    // --- All valves confirmed off
    logs.M_LogInfo('LN2 filling stopped successfully.');
    M_Activity_Stop_LN2_Filling := TRUE;
    TurningOFFTimeout(IN := FALSE);
    bAttemptingTurnOFF := FALSE;
    RETURN;
ELSE
    // --- Timeout expired: check what remains active
    IF lc_ln2_level_ctrl[1].LN2_Valve.stat.bActive THEN
        logs.M_LogInfo('LN2 shutdown timeout – Valve 1 still active');
        M_SetError(E1207_LN2_SHUTDOWN_V1_FAILED, 'LN2 Valve 1 failed to turn off');
    END_IF
    IF lc_ln2_level_ctrl[2].LN2_Valve.stat.bActive THEN
        logs.M_LogInfo('LN2 shutdown timeout – Valve 2 still active');
        M_SetError(E1208_LN2_SHUTDOWN_V2_FAILED, 'LN2 Valve 2 failed to turn off');
    END_IF
    IF lc_ln2_level_ctrl[3].LN2_Valve.stat.bActive THEN
        logs.M_LogInfo('LN2 shutdown timeout – Valve 3 still active');
        M_SetError(E1209_LN2_SHUTDOWN_V3_FAILED, 'LN2 Valve 3 failed to turn off');
    END_IF

    IF lc_ln2_level_ctrl[1].LN2_Valve.stat.bActive
    OR lc_ln2_level_ctrl[2].LN2_Valve.stat.bActive
    OR lc_ln2_level_ctrl[3].LN2_Valve.stat.bActive THEN
        M_SetError(E1206_LN2_Level_ShutdownTimeout, 'LN2 shutdown timeout: one or more valves still active');
        TurningOFFTimeout(IN := FALSE);
        bAttemptingTurnOFF := FALSE;
        M_Activity_Stop_LN2_Filling := FALSE;
        RETURN;
    ELSE
        logs.M_LogInfo('LN2 filling turned off successfully (after timeout).');
        M_Activity_Stop_LN2_Filling := TRUE;
        TurningOFFTimeout(IN := FALSE);
        bAttemptingTurnOFF := FALSE;
        RETURN;
    END_IF
END_IF
END_METHOD

METHOD M_Activity_Stop_PTCs : BOOL
VAR_INPUT
END_VAR
VAR_INST
    bErrorCond            : BOOL := FALSE;
    bAttemptingTurnOFF    : BOOL := FALSE;

    TurningOFFTimeout     : TON;
    tTurningOFFTime       : TIME := T#10M;
END_VAR
//  Start shutdown process 
IF NOT bAttemptingTurnOFF THEN
    bAttemptingTurnOFF := TRUE;
    logs.M_LogInfo('Initiating PTC shutdown...');
    
    TurningOFFTimeout(IN := TRUE, PT := tTurningOFFTime);
	ctrl.bPTC_1_Enable := FALSE;
	ctrl.bPTC_2_Enable := FALSE;
	ctrl.bPTC_3_Enable := FALSE;
END_IF

// Wait for confirmation of shutdown or timeout
IF NOT TurningOFFTimeout.Q THEN
    IF ptc[1].stat.bSystemOn OR ptc[2].stat.bSystemOn OR ptc[3].stat.bSystemOn THEN
        M_Activity_Stop_PTCs := FALSE;
        RETURN;
    END_IF

    // All PTCs confirmed off
    logs.M_LogInfo('PTCs successfully turned off.');
    M_Activity_Stop_PTCs := TRUE;
    TurningOFFTimeout(IN := FALSE);
    bAttemptingTurnOFF := FALSE;
    RETURN;
ELSE
    // Timeout expired — check if PTC or PTCs are still active
    IF ptc[1].stat.bSystemOn OR ptc[2].stat.bSystemOn OR ptc[3].stat.bSystemOn THEN
        logs.M_LogInfo('PTC shutdown timeout – one or more PTCs failed to stop.');
        M_SetError(E1907_PTC_ShutdownTimeout, 'PTC shutdown timeout: at least one PTC still active.');
        TurningOFFTimeout(IN := FALSE);
        bAttemptingTurnOFF := FALSE;
        M_Activity_Stop_PTCs := FALSE;
        RETURN;
    ELSE
        logs.M_LogInfo('PTCs turned off successfully (after timeout).');
        M_Activity_Stop_PTCs := TRUE;
        TurningOFFTimeout(IN := FALSE);
        bAttemptingTurnOFF := FALSE;
        RETURN;
    END_IF
END_IF
END_METHOD

METHOD M_Activity_Stopping_Cool_Down : BOOL
VAR_INPUT
END_VAR
VAR_IN_OUT
	{attribute 'OPC.UA.DA' := '0'}
	all_cryo_temps:					FB_METIS_TEMPERATURES;
	{attribute 'OPC.UA.DA' := '0'}
	all_heaters:					FB_METIS_HEATERS;
	{attribute 'OPC.UA.DA' := '0'}
	all_t_ctrls:      				FB_METIS_TCTRL;
	{attribute 'OPC.UA.DA' := '0'}
	all_t_votes: 					FB_METIS_VOTERS;
	{attribute 'OPC.UA.DA' := '0'}
	interlocks:						T_METIS_CRYO_INTERLOCKS;
END_VAR
VAR_INST
    StopCooldownAttempts : UINT := 0;
    MaxStopCooldownAttempts : UINT := 3; 
END_VAR
CASE stat.nStopCoolDownState OF

// Check readiness 
0:
    logs.M_LogInfo('Stopping cooldown: checking if system is ready for operation...');
    
    IF stat.bReadyForOperations THEN
		
		stat.bPermitEvacuationStop := TRUE;
        M_PermitEvacuationStop();
        logs.M_LogInfo('System is cold and ready – evacuation stop permitted.');
        stat.nStopCoolDownState := 50;

    ELSE
		stat.bPermitEvacuationStop := FALSE;
        logs.M_LogInfo('System is not cold – evacuation stop blocked.');
		// stat.nState := E_MET_CRYO_COOLDOWN_STATE.KEEP_COOLING;
		//M_Activity_Stopping_Cool_Down := FALSE;
        stat.nStopCoolDownState := 50;
    END_IF
    

// Declare Cooldown Finished
50:
    logs.M_LogInfo('Cooldown process finished.');
    stat.nState := E_MET_CRYO_COOLDOWN_STATE.FINISHED;
    stat.nStopCoolDownState := 0; 
    M_Activity_Stopping_Cool_Down := TRUE;
    RETURN;

// Error state 
99:
    logs.M_LogInfo('Cooldown stop failed. Entered error fallback.');
    stat.nState := E_MET_CRYO_COOLDOWN_STATE.ERROR;
    M_Activity_Stopping_Cool_Down := FALSE;
    RETURN;

END_CASE

M_Activity_Stopping_Cool_Down := FALSE;
END_METHOD

METHOD M_Check_Is_ReadyForOperation : BOOL
VAR_INPUT
END_VAR
VAR_IN_OUT
	{attribute 'OPC.UA.DA' := '0'}
	all_cryo_temps:					FB_METIS_TEMPERATURES;
	{attribute 'OPC.UA.DA' := '0'}
	all_heaters:					FB_METIS_HEATERS;
	{attribute 'OPC.UA.DA' := '0'}
	all_t_ctrls:      				FB_METIS_TCTRL;
	{attribute 'OPC.UA.DA' := '0'}
	all_t_votes: 					FB_METIS_VOTERS;
	{attribute 'OPC.UA.DA' := '0'}
	interlocks:						T_METIS_CRYO_INTERLOCKS;
END_VAR
// Check if the system is ready for operations (all temps achieved)




IF in_Cryo_Stat.bInGoodVacuum AND in_Cryo_Stat.lrRadiationShieldsTempK <  100.0 AND in_Cryo_Stat.lrHighestTempK < 75.0 THEN
	stat.bReadyForOperations := TRUE;
ELSE
	stat.bReadyForOperations := FALSE;
END_IF
END_METHOD

METHOD M_Check_LN2_Filling_Status : BOOL
VAR_INPUT
END_VAR
VAR_INST
	bLN2_FillingError :		BOOL := TRUE;
	bAttemptingRecovery:	BOOL := FALSE;
	RecoveryTimeout:		TON;
	tRecoveryTime:			TIME := T#30S;
END_VAR
// precondition checks

bLN2_FillingError := FALSE;

IF NOT in_Cryo_Stat.bEvacuationActive THEN
    IF NOT bLN2_FillingError THEN
        M_SetError(E1004_PumpsNotRunning, 'Evacuation is not active');
        bLN2_FillingError := TRUE;
    END_IF
ELSIF NOT bESO_LN2_Supply THEN
    IF NOT bLN2_FillingError THEN
        M_SetError(E1005_LN2SupplyNotReady, 'LN2 supply unavailable');
        bLN2_FillingError := TRUE;
    END_IF
END_IF

// Valve error checks
IF lc_ln2_level_ctrl[1].LN2_Valve.stat.bError THEN
    M_SetError(E1100_SHA_V_Error, 'Error in LN2 Valve – Stiff Ring');
    bLN2_FillingError := TRUE;
ELSIF lc_ln2_level_ctrl[2].LN2_Valve.stat.bError THEN
    M_SetError(E1101_SHB_V_Error, 'Error in LN2 Valve – Middle Segment');
    bLN2_FillingError := TRUE;
ELSIF lc_ln2_level_ctrl[3].LN2_Valve.stat.bError THEN
    M_SetError(E1102_SHC_V_Error, 'Error in LN2 Valve – Lower Segment');
    bLN2_FillingError := TRUE;
END_IF

//IF NOT lc_ln2_level_ctrl[1].bActive OR NOT lc_ln2_level_ctrl[2].bActive OR NOT lc_ln2_level_ctrl[3].bActive THEN
//	 bLN2_FillingError := TRUE;
//END_IF

// Recoverying
IF NOT bLN2_FillingError THEN
	
	// All is good
	RecoveryTimeout(IN := FALSE);
	bAttemptingRecovery := FALSE;
	bLN2_FillingError := FALSE;
	M_Check_LN2_Filling_Status := TRUE;
	RETURN;
ELSE

    IF NOT bAttemptingRecovery THEN
        bAttemptingRecovery := TRUE;
        RecoveryTimeout(IN := TRUE, PT := tRecoveryTime);
		logs.M_LogInfo('Error LN2 Filling: Recovering...');
		ctrl.bEnable_LN2_Level_Control[1] := FALSE;
		ctrl.bEnable_LN2_Level_Control[2] := FALSE;
		ctrl.bEnable_LN2_Level_Control[3] := FALSE;
		lc_ln2_level_ctrl[1].LN2_Valve.M_Reset();
        lc_ln2_level_ctrl[2].LN2_Valve.M_Reset();
        lc_ln2_level_ctrl[3].LN2_Valve.M_Reset();
		lc_ln2_level_ctrl[1].M_Reset();
		lc_ln2_level_ctrl[2].M_Reset();
		lc_ln2_level_ctrl[3].M_Reset();
    END_IF

    IF NOT RecoveryTimeout.Q THEN
		ctrl.bEnable_LN2_Level_Control[1] := TRUE;
		ctrl.bEnable_LN2_Level_Control[2] := TRUE;
		ctrl.bEnable_LN2_Level_Control[3] := TRUE;
		RecoveryTimeout(IN := TRUE, PT := tRecoveryTime);
    ELSE
        // Recovery failed → shutdown filling
        ctrl.bEnable_LN2_Level_Control[1] := FALSE;
        ctrl.bEnable_LN2_Level_Control[2] := FALSE;
        ctrl.bEnable_LN2_Level_Control[3] := FALSE;
        tDelay_SHB(IN := FALSE);
        tDelay_SHC(IN := FALSE);
        stat.nState := E_MET_CRYO_COOLDOWN_STATE.ERROR;
        stat.sState := 'LN2 Filling Failed – Recovery Timeout';
		logs.M_LogInfo('LN2 Filling Failed – Recovery Timeout');
        RecoveryTimeout(IN := FALSE);
        bAttemptingRecovery := FALSE;
    END_IF

    M_Check_LN2_Filling_Status := FALSE;
    RETURN;
END_IF
END_METHOD

METHOD M_Check_PTCs_Heater_Ctrl_Status : BOOL
VAR_INPUT
END_VAR
VAR_INST
    bErrorCond           : BOOL := FALSE;
    bAttemptingRecovery  : BOOL := FALSE;	
END_VAR
VAR_IN_OUT
	{attribute 'OPC.UA.DA' := '0'}
	all_cryo_temps:					FB_METIS_TEMPERATURES;
	{attribute 'OPC.UA.DA' := '0'}
	all_heaters:					FB_METIS_HEATERS;
	{attribute 'OPC.UA.DA' := '0'}
	all_t_ctrls:      				FB_METIS_TCTRL;
	{attribute 'OPC.UA.DA' := '0'}
	all_t_votes: 					FB_METIS_VOTERS;
	{attribute 'OPC.UA.DA' := '0'}
	interlocks:						T_METIS_CRYO_INTERLOCKS;
END_VAR


IF 	all_heaters.h_cry_pta.stat.bError THEN
	M_SetError(E1308_EarFlange_TempCtrlFault, 'h_cry_pta in error...');
    bErrorCond := TRUE;
END_IF

IF 	all_heaters.h_cry_ptb.stat.bError THEN
	M_SetError(E1308_EarFlange_TempCtrlFault, 'h_cry_ptb in error...');
    bErrorCond := TRUE;
END_IF

IF 	all_heaters.h_cry_ptc.stat.bError THEN
	M_SetError(E1308_EarFlange_TempCtrlFault, 'h_cry_ptc in error...');
    bErrorCond := TRUE;
END_IF

IF 	all_t_ctrls.tc_cry_pt.stat.bError THEN
	M_SetError(E1308_EarFlange_TempCtrlFault, 'tc_cry_pt temp ctrl in error...');
    bErrorCond := TRUE;
END_IF


IF bErrorCond THEN
	
	M_Check_PTCs_Heater_Ctrl_Status := FALSE;
	logs.M_LogInfo('Temp Ctrl anomaly at stiff ring');
	stat.bWarning := TRUE;
    RETURN;
	
END_IF


M_Check_PTCs_Heater_Ctrl_Status := TRUE;
END_METHOD

METHOD M_Check_PTCs_Status : BOOL
VAR_INPUT
END_VAR
VAR_INST
    bErrorCond           : BOOL := FALSE;
    bAttemptingRecovery  : BOOL := FALSE;

    RecoveryTimeout      : TON;
    tRecoveryTime        : TIME := T#10M;

    ToggleTimeoutPTC1    : TON;
    ToggleTimeoutPTC2    : TON;
    ToggleTimeoutPTC3    : TON;
    tToggleTime          : TIME := T#5M;

    bTogglePTC1          : BOOL := FALSE;
    bTogglePTC2          : BOOL := FALSE;
    bTogglePTC3          : BOOL := FALSE;
END_VAR


// Check PTC Active Status
bErrorCond := FALSE;

IF NOT ptc[1].stat.bActive THEN
    M_SetError(E1903_PTC1_NotActive, 'PTC 1 not active');
    bErrorCond := TRUE;
END_IF

IF NOT ptc[2].stat.bActive THEN
    M_SetError(E1904_PTC2_NotActive, 'PTC 2 not active');
    bErrorCond := TRUE;
END_IF

IF NOT ptc[3].stat.bActive THEN
    M_SetError(E1905_PTC3_NotActive, 'PTC 3 not active');
    bErrorCond := TRUE;
END_IF

IF NOT bErrorCond THEN
    RecoveryTimeout		(IN := FALSE);
    ToggleTimeoutPTC1	(IN := FALSE);
    ToggleTimeoutPTC2	(IN := FALSE);
    ToggleTimeoutPTC3	(IN := FALSE);
    bAttemptingRecovery := FALSE;
    M_Check_PTCs_Status := TRUE;
    RETURN;
END_IF

// Handle Recovery
IF NOT bAttemptingRecovery THEN
    bAttemptingRecovery := TRUE;
    RecoveryTimeout(IN := TRUE, PT := tRecoveryTime);
    logs.M_LogInfo('PTC failure detected: entering recovery...');
END_IF

IF NOT RecoveryTimeout.Q THEN

    //  PTC 1 Recovery Toggle
    IF NOT ptc[1].stat.bActive THEN
        ToggleTimeoutPTC1(IN := TRUE, PT := tToggleTime);
        IF ToggleTimeoutPTC1.Q THEN
            IF bTogglePTC1 THEN
                ptc[1].in_bEnable := TRUE;
            ELSE
                ptc[1].in_bEnable := FALSE;
            END_IF
            bTogglePTC1 := NOT bTogglePTC1;
            ToggleTimeoutPTC1(IN := FALSE); // Restart toggle delay
        END_IF
    ELSE
        ToggleTimeoutPTC1(IN := FALSE);
    END_IF

    // PTC 2 Recovery Toggle
    IF NOT ptc[2].stat.bActive THEN
        ToggleTimeoutPTC2(IN := TRUE, PT := tToggleTime);
        IF ToggleTimeoutPTC2.Q THEN
            IF bTogglePTC2 THEN
                ptc[2].in_bEnable := TRUE;
            ELSE
                ptc[2].in_bEnable := FALSE;
            END_IF
            bTogglePTC2 := NOT bTogglePTC2;
            ToggleTimeoutPTC2(IN := FALSE);
        END_IF
    ELSE
        ToggleTimeoutPTC2(IN := FALSE);
    END_IF

    // PTC 3 Recovery Toggle
    IF NOT ptc[3].stat.bActive THEN
        ToggleTimeoutPTC3(IN := TRUE, PT := tToggleTime);
        IF ToggleTimeoutPTC3.Q THEN
            IF bTogglePTC3 THEN
                ptc[3].in_bEnable := TRUE;
            ELSE
                ptc[3].in_bEnable := FALSE;
            END_IF
            bTogglePTC3 := NOT bTogglePTC3;
            ToggleTimeoutPTC3(IN := FALSE);
        END_IF
    ELSE
        ToggleTimeoutPTC3(IN := FALSE);
    END_IF

    M_Check_PTCs_Status := FALSE;
    RETURN;
ELSE
    // Recovery Failed 
    ptc[1].in_bEnable := FALSE;
    ptc[2].in_bEnable := FALSE;
    ptc[3].in_bEnable := FALSE;

    stat.bWarning := TRUE;
    M_SetError(E1906_PTC_Failure, 'PTC recovery failed after timeout');
    stat.nState := E_MET_CRYO_COOLDOWN_STATE.STOPPING_COOL_DOWN;
    RecoveryTimeout(IN := FALSE);
    ToggleTimeoutPTC1(IN := FALSE);
    ToggleTimeoutPTC2(IN := FALSE);
    ToggleTimeoutPTC3(IN := FALSE);

    bAttemptingRecovery := FALSE;
    M_Check_PTCs_Status := FALSE;
END_IF
END_METHOD

METHOD M_Configure
VAR_INPUT
END_VAR

	////////////////////////
	// Pre-Cooling valves//
	//////////////////////



// Set pointers to Valves - MUST!!!
ptrV[1]	:= ADR(PVV_P1);
ptrV[2]	:= ADR(PVV_P2);
ptrV[3]	:= ADR(PVV_P3);


// Set pointers to Valve Commands - MUST!!!
ptrVC[1]	:= ADR(ctrl.cor_PVV_P1);
ptrVC[2]	:= ADR(ctrl.cor_PVV_P2);
ptrVC[3]	:= ADR(ctrl.cor_PVV_P3);


// Set pointers to Enable Valves flags - MUST!!!
ptrEV[1]	:= ADR(ctrl.bEnable_PVV_P1);
ptrEV[2]	:= ADR(ctrl.bEnable_PVV_P2);
ptrEV[3]	:= ADR(ctrl.bEnable_PVV_P3);



IF NOT bConfigured THEN


	bPwr_VAG_PCA 	:= TRUE;
	bPwr_VAG_PCB 	:= TRUE;      
	bPwr_VAG_P1 	:= TRUE;
	
	PVV_P1.M_Reset();
	PVV_P2.M_Reset();
	PVV_P3.M_Reset();
	
	///////////////////////
	///// PTC Coolers /////
	//////////////////////		

	// Set pointers to command override instances
	ptrArr_cor_ptcs[1] := ADR(ctrl.cor_PTC_1);
	ptrArr_cor_ptcs[2] := ADR(ctrl.cor_PTC_2);
	ptrArr_cor_ptcs[3] := ADR(ctrl.cor_PTC_3);
	
	
	////////////////////////////////
	// LN2 Level Sensors & Control//
	////////////////////////////////

	ctrl.bEnable_LN2_Level_Control[1] := FALSE;
	ctrl.bEnable_LN2_Level_Control[2] := FALSE;
	ctrl.bEnable_LN2_Level_Control[3] := FALSE; 
	
	
	// This call just configures logs at the very start.
	// Logging is done by explicit calls to M_LogInfo().
	logs(in_sName := in_sName);
	
	M_ResetValves();
	
	bConfigured := TRUE;

END_IF
END_METHOD

METHOD M_ExecuteControllers
VAR_INPUT
END_VAR
////////////////////////
// Pre-Cooling valves//
//////////////////////

//ctrl.bEnable_PVV_P1 := in_bEnable_PVV_P1;
ctrl.bEnable_PVV_P1 := TRUE; // TODO: Implement for EVAC and Pre-cooling
ctrl.bEnable_PVV_P2 := in_bEnable_PVV_P2;
ctrl.bEnable_PVV_P3 := in_bEnable_PVV_P3;

// Valve commands
ctrl.cor_PVV_P1(in_bEnable := ctrl.bEnable_PVV_P1);	// Handling of PVV_P1 commands
ctrl.cor_PVV_P2(in_bEnable := ctrl.bEnable_PVV_P2);	// Handling of PVV_P2 commands
ctrl.cor_PVV_P3(in_bEnable := ctrl.bEnable_PVV_P3);	// Handling of PVV_P3 commands

// Valve Control
IF PVV_P1.stat.bError THEN
	PVV_P1.M_Reset();
END_IF 
PVV_P1(
	in_bEnable			:= ctrl.cor_PVV_P1.out_bEnable,
	in_nFeedback		:= E_CRYO_BIN_ACT_FEEDBACK.ON_AND_OFF);
	
PVV_P2(
	in_bEnable			:= ctrl.cor_PVV_P2.out_bEnable,
	in_nFeedback		:= E_CRYO_BIN_ACT_FEEDBACK.ON_AND_OFF);
	
PVV_P3(
	in_bEnable			:= ctrl.cor_PVV_P3.out_bEnable,
	in_nFeedback		:= E_CRYO_BIN_ACT_FEEDBACK.ON_AND_OFF);


///////////////////////
// LN2 Level Sensors//
//////////////////////



lc_ln2_level_ctrl[1](in_sName := 'Stiff_Ring',
					in_bEnable:= ctrl.bEnable_LN2_Level_Control[1], 
					in_ESO_LN2_Supply := bESO_LN2_Supply,
					in_bEarly_Refilling:= FALSE);
	
lc_ln2_level_ctrl[2](in_sName := 'Intermediate_Segment',
					in_bEnable:= ctrl.bEnable_LN2_Level_Control[2], 
					in_ESO_LN2_Supply := bESO_LN2_Supply,
					in_bEarly_Refilling:= FALSE);

lc_ln2_level_ctrl[3](in_sName := 'Bottom_Segment',
					in_bEnable:= ctrl.bEnable_LN2_Level_Control[3], 
					in_ESO_LN2_Supply := bESO_LN2_Supply,
					in_bEarly_Refilling:= FALSE);
	
	
///////////////////////
///// PTC Coolers /////
//////////////////////	

{IF defined (V1_HW)}
	
ctrl.cor_PTC_1(in_bEnable:=ctrl.bPTC_1_Enable);
ptc[1](
	in_bEnable:= ctrl.cor_PTC_1.out_bEnable,
	in_bSimulation:= FALSE, 
	in_sName:= 'PTC_A', 
	in_sSN_Compressor:= 'CPA286IW-19880300001', 
	in_sSN_PulseTube:= 'PT810-19880200001', 
	in_nYear_Compressor:= 2023, 
	in_nYear_PulseTube:= 2023, 
	in_lrNextService_Compressor:= 20000.0, 
	in_lrNextService_PulseTube:= 40000.0, 
	in_nSlaveID:= 16, 
	in_nPeriod:= 1000);
	

ctrl.cor_PTC_2(in_bEnable:=ctrl.bPTC_2_Enable);
ptc[2](
	in_bEnable:= ctrl.cor_PTC_2.out_bEnable,
	in_bSimulation:= FALSE, 
	in_sName:= 'PTC_B', 
	in_sSN_Compressor:= 'CPA286IW-19870300001', 
	in_sSN_PulseTube:= 'PT810-19870200001', 
	in_nYear_Compressor:= 2023, 
	in_nYear_PulseTube:= 2023, 
	in_lrNextService_Compressor:= 20000.0, 
	in_lrNextService_PulseTube:= 40000.0, 
	in_nSlaveID:= 16, 
	in_nPeriod:= 1000);
	

ctrl.cor_PTC_3(in_bEnable:=ctrl.bPTC_3_Enable);
ptc[3](
	in_bEnable:= ctrl.cor_PTC_3.out_bEnable,
	in_bSimulation:= FALSE, 
	in_sName:= 'PTC_C', 
	in_sSN_Compressor:= 'CPA286IW-19890300001', 
	in_sSN_PulseTube:= 'PT810-19890200001', 
	in_nYear_Compressor:= 2023, 
	in_nYear_PulseTube:= 2023, 
	in_lrNextService_Compressor:= 20000.0, 
	in_lrNextService_PulseTube:= 40000.0, 
	in_nSlaveID:= 16, 
	in_nPeriod:= 1000);

{END_IF}
 
{IF defined (V2_SIM)}	
	
ctrl.cor_PTC_1(in_bEnable:=ctrl.bPTC_1_Enable);
ptc[1](
	in_bEnable:= ctrl.cor_PTC_1.out_bEnable,
	in_bSimulation:= FALSE, 
	in_sName:= 'PTC_A', 
	in_sSN_Compressor:= 'CPA286IW-19880300001', 
	in_sSN_PulseTube:= 'PT810-19880200001', 
	in_nYear_Compressor:= 2023, 
	in_nYear_PulseTube:= 2023, 
	in_lrNextService_Compressor:= 20000.0, 
	in_lrNextService_PulseTube:= 40000.0, 
	in_nSlaveID:= 16, 
	in_nPeriod:= 1000);
	

ctrl.cor_PTC_2(in_bEnable:=ctrl.bPTC_2_Enable);
ptc[2](
	in_bEnable:= ctrl.cor_PTC_2.out_bEnable,
	in_bSimulation:= TRUE, 
	in_sName:= 'PTC_B', 
	in_sSN_Compressor:= 'CPA286IW-19870300001', 
	in_sSN_PulseTube:= 'PT810-19870200001', 
	in_nYear_Compressor:= 2023, 
	in_nYear_PulseTube:= 2023, 
	in_lrNextService_Compressor:= 20000.0, 
	in_lrNextService_PulseTube:= 40000.0, 
	in_nSlaveID:= 16, 
	in_nPeriod:= 1000);
	

ctrl.cor_PTC_3(in_bEnable:=ctrl.bPTC_3_Enable);
ptc[3](
	in_bEnable:= ctrl.cor_PTC_3.out_bEnable,
	in_bSimulation:= FALSE, 
	in_sName:= 'PTC_C', 
	in_sSN_Compressor:= 'CPA286IW-19890300001', 
	in_sSN_PulseTube:= 'PT810-19890200001', 
	in_nYear_Compressor:= 2023, 
	in_nYear_PulseTube:= 2023, 
	in_lrNextService_Compressor:= 20000.0, 
	in_lrNextService_PulseTube:= 40000.0, 
	in_nSlaveID:= 16, 
	in_nPeriod:= 1000);	
		
	
{END_IF}	
	
///////////////////////
///// ---------- /////
//////////////////////
END_METHOD

METHOD M_Get_ReadyForOperations : BOOL
VAR_INPUT
END_VAR
M_Get_ReadyForOperations := stat.bReadyForOperations;
END_METHOD

METHOD M_HandleEvents
VAR_INPUT
END_VAR

//
// Handle triggers
//

trigEnable	(CLK := ctrl.bEnable);
trigDisable	(CLK := ctrl.bEnable);
END_METHOD

METHOD M_HandleInterlocks
VAR_INPUT
END_VAR
//VAR_IN_OUT
//	{attribute 'OPC.UA.DA' := '0'}
//	interlocks:						T_METIS_CRYO_INTERLOCKS;
//END_VAR

//interlocks.bInterlock_Evacuation 			:= FALSE;
//interlocks.bInterlock_Venting 			:= TRUE; // Venting blocked
//interlocks.bInterlock_CoolDown 			:= FALSE; // Cool_Down, pre-cooling, LN2_filling blocked
//interlocks.bInterlock_WarmUp 				:= TRUE; // Warm_up Blocked
//interlocks.bInterlock_Regeneration 		:= TRUE;
//interlocks.bInterlock_AntiFogging 		:= FALSE;
//interlocks.bInterlock_PowerOutage 		:= FALSE;
//interlocks.bInterlock_StopPowerOutage		:= FALSE;

//interlocks.sInterlockState := 'COOL_DOWN Active';



//// Venting Valves Closed ---
//IF in_Cryo_Stat.bVentingValvesAreClosed THEN
//    stat.nState := E_MET_CRYO_VENTING_STATE.ERROR;
//    stat.sState := 'Error: Venting valves are closed.';
//    RETURN; 
//END_IF

//// Pumps Running ---
//IF in_Cryo_Stat.bPumpsAreRunning THEN
//    stat.nState := E_MET_CRYO_VENTING_STATE.ERROR;
//    stat.sState := 'Error: Pumps are Running.';
//    RETURN; 
//END_IF

//// --- Evacuation Activated ---
//IF in_Cryo_Stat.bEvacuationActive THEN
//    stat.nState := E_MET_CRYO_VENTING_STATE.ERROR;
//    stat.sState := 'Error: Evacuation Activated.';
//    RETURN; 
//END_IF

//// --- Cool Down Active ---
//IF in_Cryo_Stat.bCoolDownActive THEN
//    stat.nState := E_MET_CRYO_VENTING_STATE.ERROR;
//    stat.sState := 'Error: Cool down activated.';
//    RETURN; 
//END_IF

//// --- Regeneration Active ---
//IF in_Cryo_Stat.bRegenerationActive THEN
//    stat.nState := E_MET_CRYO_VENTING_STATE.ERROR;
//    stat.sState := 'Error: Regeneration activated.';
//    RETURN; 
//END_IF

//// --- GN2 supply disconnected ---
//IF NOT in_Cryo_Stat.bGN2SupplyConnected THEN
//    stat.nState := E_MET_CRYO_VENTING_STATE.ERROR;
//    stat.sState := 'Error: GN2 supply  disconnected.';
//    RETURN; 
//END_IF

//IF HPG.stat.lrPressure > (cfg.lrMaxVentingPressure + 10) THEN
//    stat.nState := E_MET_CRYO_VENTING_STATE.ERROR;
//    stat.sState := 'Error: Pressure in vessle too high';
//	(*TODO: Implement critical Alarm*)
//    RETURN;
//END_IF
END_METHOD

METHOD M_Manage_Early_Refilling : BOOL
VAR_INPUT
END_VAR
VAR
    bAllHighReached : BOOL;
END_VAR


M_Manage_Early_Refilling := FALSE;


CASE stat.nState OF

    // *********************************
    // Allowed "active" states:
    // Early refilling logic may run / continue here
    // ***********************************************
    E_MET_CRYO_COOLDOWN_STATE.START_FILLING_LN2,
    E_MET_CRYO_COOLDOWN_STATE.START_PTCS,
    E_MET_CRYO_COOLDOWN_STATE.START_TEMP_CTRL_PTC,
    E_MET_CRYO_COOLDOWN_STATE.KEEP_COOLING:
        
        // 1) Latch "HIGH level reached at least once" for each vessel
        IF lc_ln2_level_ctrl[1].out_LN2_Level = E_METIS_CRYO_LN2_SENSOR_LEVELS.HIGH THEN
            bHighReachedSHA := TRUE;
        END_IF

        IF lc_ln2_level_ctrl[2].out_LN2_Level = E_METIS_CRYO_LN2_SENSOR_LEVELS.HIGH THEN
            bHighReachedSHB := TRUE;
        END_IF

        IF lc_ln2_level_ctrl[3].out_LN2_Level = E_METIS_CRYO_LN2_SENSOR_LEVELS.HIGH THEN
            bHighReachedSHC := TRUE;
        END_IF

        bAllHighReached := bHighReachedSHA AND bHighReachedSHB AND bHighReachedSHC;
		

        // 2) Once all HIGH levels have been reached at least once,
        //    start early refilling (only once)
        IF bAllHighReached AND NOT bEarlyRefillingActive THEN
            bEarlyRefillingActive := TRUE;
            bRestartCycle := FALSE;
			
			stat.sEarlyFillState := 'Early Refilling Started';			

            // Start the 24-hour total timer
            tonEarlyRefillTotal(IN := TRUE, PT := tEarlyRefillTotal);

            // Start the 2-hour cycle timer
            tonEarlyRefillCycle(IN := TRUE, PT := tEarlyRefillCycle);
		ELSE
			stat.sEarlyFillState := 'Early Refilling Started: Waiting High level on all vessels at least once';
        END_IF

        // 3) If early refilling is active, manage timers and refilling cycles
        IF bEarlyRefillingActive THEN

            // Keep 24-hour timer running
            tonEarlyRefillTotal(IN := TRUE, PT := tEarlyRefillTotal);

            // Handle the 2-hour cycle between refills
            IF NOT bRestartCycle THEN
                // Normal timing phase: run the 2-hour timer
                tonEarlyRefillCycle(IN := TRUE, PT := tEarlyRefillCycle);

                IF tonEarlyRefillCycle.Q THEN
                    // 2 hours elapsed -> start refilling on all three vessels
                    lc_ln2_level_ctrl[1].M_Set_LN2FillingFlag();
                    lc_ln2_level_ctrl[2].M_Set_LN2FillingFlag();
                    lc_ln2_level_ctrl[3].M_Set_LN2FillingFlag();

                    // Next cycle: reset the timer once
                    bRestartCycle := TRUE;
                END_IF
            ELSE
                // Reset the 2-hour timer once, then return to timing mode
                tonEarlyRefillCycle(IN := FALSE, PT := tEarlyRefillCycle);

                IF NOT tonEarlyRefillCycle.Q THEN
                    bRestartCycle := FALSE;
                END_IF
            END_IF

            // 4) Stop condition for early refilling:
            //    - 24 hours elapsed, or
            //    - external disable trigger fired (trigDisable.Q = TRUE)
            IF tonEarlyRefillTotal.Q OR trigDisable.Q THEN
                bEarlyRefillingActive := FALSE;

                tonEarlyRefillTotal(IN := FALSE, PT := tEarlyRefillTotal);
                tonEarlyRefillCycle(IN := FALSE, PT := tEarlyRefillCycle);

                bRestartCycle := FALSE;

                // Early refilling period completed or cancelled
                M_Manage_Early_Refilling := TRUE;
				bEarlyRefillDone := TRUE;
				stat.sEarlyFillState := 'Early Refilling Finished.';
				stat.sEarlyFillSubState := '';
            END_IF
			
			stat.sEarlyFillState := CONCAT('Early refilling duration: ',
							 F_TON_TO_TIME_STRING(Timer := tonEarlyRefillTotal));
			stat.sEarlyFillSubState := CONCAT('Refilling cycle: ',
							 F_TON_TO_TIME_STRING(Timer := tonEarlyRefillCycle));
        END_IF


    // ------------------------------------------------------
    // STOPPING_COOL_DOWN:
    // Early refilling must stop here (cleanup only)
    // ------------------------------------------------------
    E_MET_CRYO_COOLDOWN_STATE.STOPPING_COOL_DOWN:

        // Stop early refilling and reset timers
        bEarlyRefillingActive := FALSE;

        tonEarlyRefillTotal(IN := FALSE, PT := tEarlyRefillTotal);
        tonEarlyRefillCycle(IN := FALSE, PT := tEarlyRefillCycle);

        bRestartCycle := FALSE;

        // Do not change the HIGH-reached latches here (can be useful diagnostically)
        // Signal that early refilling is finished with respect to this activity
        M_Manage_Early_Refilling := TRUE;
		bEarlyRefillDone := TRUE;


    // All other states:
    // NONE, CHECK_PRECONDITIONS, START_COOL_DOWN, FINISHED, ERROR
    // -> do NOTHING

    ELSE
			stat.sEarlyFillState := 'Early filling Not Active';
END_CASE
END_METHOD

METHOD M_PermitEvacuationStop : BOOL
//VAR_INPUT
//	bPermitEvacuationStop : BOOL;
//END_VAR
M_PermitEvacuationStop := stat.bPermitEvacuationStop;
END_METHOD

METHOD M_ReadSensors
VAR_INPUT
END_VAR



sensor_VAG_PCA(in_sName:= 'VAG_PCA', in_nType:= E_CRYO_SENSOR_TYPE_PRESS.PKR_360, in_lrBitsPerVolt:= , in_nSampleTime:= 100);
sensor_VAG_PCB(in_sName:= 'VAG_PCB', in_nType:= E_CRYO_SENSOR_TYPE_PRESS.PKR_360, in_lrBitsPerVolt:= , in_nSampleTime:= 100);
sensor_VAG_P1(in_sName:= 'VAG_P1', in_nType:= E_CRYO_SENSOR_TYPE_PRESS.PKR_360, in_lrBitsPerVolt:= , in_nSampleTime:= 100);


ctrl.por_VAG_PCA(in_bEnable := ctrl.bSim_Press_VAG_PCA);	// Simulation flag override
VAG_PCA(
	in_sName		:= 'VAG_PCA',
	in_bSimulation	:= ctrl.por_VAG_PCA.out_bEnable,
	in_nNumSensor	:= 2,
	in_nVoteMethod	:= E_CRYO_VOTE.V_1oo2,
	in_pSensor1		:= ADR(sensor_VAG_PCA));

ctrl.por_VAG_PCB(in_bEnable := ctrl.bSim_Press_VAG_PCB);	// Simulation flag override
VAG_PCB(
	in_sName		:= 'VAG_PCB',
	in_bSimulation	:= ctrl.por_VAG_PCB.out_bEnable,
	in_nNumSensor	:= 2,
	in_nVoteMethod	:= E_CRYO_VOTE.V_1oo2,
	in_pSensor1		:= ADR(sensor_VAG_PCB));

ctrl.por_VAG_P1(in_bEnable := ctrl.bSim_Press_VAG_P1);	// Simulation flag override
VAG_P1(
	in_sName		:= 'VAG_P1',
	in_bSimulation	:= ctrl.por_VAG_P1.out_bEnable,
	in_nNumSensor	:= 2,
	in_nVoteMethod	:= E_CRYO_VOTE.V_1oo2,
	in_pSensor1		:= ADR(sensor_VAG_P1));



// For ESO Framework to read them to display on Grafana

lrLN2_Level_Sensor_1_HA_TempK := lc_ln2_level_ctrl[1].LN2_Level.Temperature_HA.stat.lrTempK;
lrLN2_Level_Sensor_1_H_TempK := lc_ln2_level_ctrl[1].LN2_Level.Temperature_H.stat.lrTempK;
lrLN2_Level_Sensor_1_L_TempK := lc_ln2_level_ctrl[1].LN2_Level.Temperature_L.stat.lrTempK;
lrLN2_Level_Sensor_1_LA_TempK := lc_ln2_level_ctrl[1].LN2_Level.Temperature_LA.stat.lrTempK;

lrLN2_Level_Sensor_2_HA_TempK := lc_ln2_level_ctrl[2].LN2_Level.Temperature_HA.stat.lrTempK;
lrLN2_Level_Sensor_2_H_TempK := lc_ln2_level_ctrl[2].LN2_Level.Temperature_H.stat.lrTempK;
lrLN2_Level_Sensor_2_L_TempK := lc_ln2_level_ctrl[2].LN2_Level.Temperature_L.stat.lrTempK;
lrLN2_Level_Sensor_2_LA_TempK := lc_ln2_level_ctrl[2].LN2_Level.Temperature_LA.stat.lrTempK;

lrLN2_Level_Sensor_3_HA_TempK := lc_ln2_level_ctrl[3].LN2_Level.Temperature_HA.stat.lrTempK;
lrLN2_Level_Sensor_3_H_TempK := lc_ln2_level_ctrl[3].LN2_Level.Temperature_H.stat.lrTempK;
lrLN2_Level_Sensor_3_L_TempK := lc_ln2_level_ctrl[3].LN2_Level.Temperature_L.stat.lrTempK;
lrLN2_Level_Sensor_3_LA_TempK := lc_ln2_level_ctrl[3].LN2_Level.Temperature_LA.stat.lrTempK;







/////////////////////////////////////////////////
//// Read individual prevacuum pressure sensors.
/////////////////////////////////////////////////
////
//// Pressure readings are averaged over 1000 ms.
////
//// Note: Pressure sensor type is configured in cfg and overwritten in M_Configure().
////       Default is Pfeiffer PKR 360 KF25.
//sensor_VAG1	(in_nType := cfg.nType_VAG1,	in_nSampleTime := 1000);
//sensor_VAG2	(in_nType := cfg.nType_VAG2,	in_nSampleTime := 1000);
//sensor_VAG3	(in_nType := cfg.nType_VAG3,	in_nSampleTime := 1000);

////////////////////////////////////////////////
//// Use voting system to calculate pressures.
////////////////////////////////////////////////
////
//// Note: VAG 1-3 have got only one sensor pressure connected !!!
////       VAG F & G have got two pressure sensors connected !
////       VAG F & G are executed at the cryo control level and passed as inputs to this FB !
////
//ctrl.por_VAG1(in_bEnable := ctrl.bSim_Press_VAG1);	// Simulation flag override
//VAG1(
//	in_bSimulation	:= ctrl.por_VAG1.out_bEnable,
//	in_nNumSensor	:= 2,
//	in_nVoteMethod	:= E_CRYO_VOTE.V_1oo2,
//	in_pSensor1		:= ADR(sensor_VAG1));

//ctrl.por_VAG2(in_bEnable := ctrl.bSim_Press_VAG2);	// Simulation flag override
//VAG2(
//	in_bSimulation	:= ctrl.por_VAG2.out_bEnable,
//	in_nNumSensor	:= 2,
//	in_nVoteMethod	:= E_CRYO_VOTE.V_1oo2,
//	in_pSensor1		:= ADR(sensor_VAG2));

//ctrl.por_VAG3(in_bEnable := ctrl.bSim_Press_VAG3);	// Simulation flag override
//VAG3(
//	in_bSimulation	:= ctrl.por_VAG3.out_bEnable,
//	in_nNumSensor	:= 2,
//	in_nVoteMethod	:= E_CRYO_VOTE.V_1oo2,
//	in_pSensor1		:= ADR(sensor_VAG3));

	
//// Copy pressure references to local variables
//VAGF	:= in_RefVAGF;
//VAGG	:= in_RefVAGG;
END_METHOD

METHOD M_ResetValves
VAR_INPUT
END_VAR

PVV_P1.M_Reset();
PVV_P2.M_Reset();
PVV_P3.M_Reset();
END_METHOD

METHOD PRIVATE M_SetError
VAR_INPUT
    nCode     : UDINT;
    sMessage  : STRING;
END_VAR


stat.Error.nCode := nCode;
stat.Error.sMessage := sMessage;
stat.bError := TRUE;
//stat.nState := E_MET_CRYO_COOLDOWN_STATE.ERROR;
END_METHOD

METHOD M_Simulated_Sens_Acts
VAR_INPUT
END_VAR

// LN2 Level sensors' temp sensors
nSim_Temp_HA_1	:= (nSim_LN2_LS_TempK[1] - 273) * 10;
nSim_Temp_H_1	:= (nSim_LN2_LS_TempK[2] - 273) * 10;
nSim_Temp_L_1	:= (nSim_LN2_LS_TempK[3] - 273) * 10;
nSim_Temp_LA_1	:= (nSim_LN2_LS_TempK[4] - 273) * 10;

nSim_Temp_HA_2	:= (nSim_LN2_LS_TempK[5] - 273) * 10;
nSim_Temp_H_2	:= (nSim_LN2_LS_TempK[6] - 273) * 10;
nSim_Temp_L_2	:= (nSim_LN2_LS_TempK[7] - 273) * 10;
nSim_Temp_LA_2	:= (nSim_LN2_LS_TempK[8] - 273) * 10;

nSim_Temp_HA_3	:= (nSim_LN2_LS_TempK[9] - 273) * 10;
nSim_Temp_H_3	:= (nSim_LN2_LS_TempK[10] - 273) * 10;
nSim_Temp_L_3	:= (nSim_LN2_LS_TempK[11] - 273) * 10;
nSim_Temp_LA_3	:= (nSim_LN2_LS_TempK[12] - 273) * 10;
END_METHOD

METHOD M_Standalone_LN2_Filling : BOOL
VAR_INPUT
END_VAR
VAR_IN_OUT
	{attribute 'OPC.UA.DA' := '0'}
	all_cryo_temps:					FB_METIS_TEMPERATURES;
	{attribute 'OPC.UA.DA' := '0'}
	all_heaters:					FB_METIS_HEATERS;
	{attribute 'OPC.UA.DA' := '0'}
	all_t_ctrls:      				FB_METIS_TCTRL;
	{attribute 'OPC.UA.DA' := '0'}
	all_t_votes: 					FB_METIS_VOTERS;
	{attribute 'OPC.UA.DA' := '0'}
	interlocks:						T_METIS_CRYO_INTERLOCKS;
END_VAR
VAR_INST
	tDelaySHB:			TIME := T#900S;
	tDelaySHC:			TIME := T#900S;
END_VAR

// IF Cool Down is not stopped manually 

IF NOT trigDisable.Q THEN 
	
		CASE stat.nStandAloneFillingState OF
	
		E_MET_CRYO_LN2_FILLING_STATE.NONE:
		
			IF bStandaloneLN2Filling THEN

				stat.nStandAloneFillingState := E_MET_CRYO_LN2_FILLING_STATE.CHECK_PRECONDITIONS; 
		
			ELSE
				
				stat.nStandAloneFillingState := E_MET_CRYO_LN2_FILLING_STATE.RADIATION_SHIELDS_COLD;
			
			END_IF
				
		(**** Preconditions check ****)
		
		E_MET_CRYO_LN2_FILLING_STATE.CHECK_PRECONDITIONS: 

			IF NOT in_Cryo_Stat.bEvacuationActive OR NOT in_Cryo_Stat.bPumpsAreRunning THEN
				M_SetError(E1004_PumpsNotRunning, 'Evacuation is not active');
				stat.nStandAloneFillingState := E_MET_CRYO_LN2_FILLING_STATE.ERROR;
			ELSIF NOT bESO_LN2_Supply THEN
				M_SetError(E1005_LN2SupplyNotReady, 'LN2 Supply is not available');
				stat.nStandAloneFillingState := E_MET_CRYO_LN2_FILLING_STATE.ERROR;
			ELSE
				stat.nStandAloneFillingState := E_MET_CRYO_LN2_FILLING_STATE.START_LEVEL_CONTROL_SHA;
				ctrl.bEnable_LN2_Level_Control[1] := TRUE; // Enable SHA control
			END_IF
			
			// Reseting LN2 level control timeouts	
			tDelay_SHB(IN := FALSE);
			tDelay_SHC(IN := FALSE);
			
			
			
		(**** Begin LN2 level control at SHA (Stiff Ring) ****)	
		
		E_MET_CRYO_LN2_FILLING_STATE.START_LEVEL_CONTROL_SHA:
		
			IF lc_ln2_level_ctrl[1].out_LN2_Level = E_METIS_CRYO_LN2_SENSOR_LEVELS.LOW OR 
				lc_ln2_level_ctrl[1].out_LN2_Level = E_METIS_CRYO_LN2_SENSOR_LEVELS.HIGH OR
				lc_ln2_level_ctrl[1].out_LN2_Level = E_METIS_CRYO_LN2_SENSOR_LEVELS.HIGH_ALARM THEN
				
				stat.nStandAloneFillingState := E_MET_CRYO_LN2_FILLING_STATE.LEVEL_LOW_SHA;
				stat.sState := 'LN2 at or above low level at SHA';
			ELSE
				
				stat.sState := 'Filling Stiff Ring...';
							
			END_IF	
			IF ctrl.bReset THEN
				stat.nStandAloneFillingState := E_MET_CRYO_LN2_FILLING_STATE.CHECK_PRECONDITIONS;
			END_IF	

		(**** LN2 reached low level at SHA ****)
		
		E_MET_CRYO_LN2_FILLING_STATE.LEVEL_LOW_SHA:
			
			tDelay_SHC(IN := TRUE, PT := tDelaySHC);
			IF tDelay_SHC.Q THEN
				// Start Bottom Segment Fill (SHC)
				ctrl.bEnable_LN2_Level_Control[3] := TRUE;
				stat.sState := 'Filling Bottom Segment...';
				stat.nStandAloneFillingState := E_MET_CRYO_LN2_FILLING_STATE.START_LEVEL_CONTROL_SHC;
				tDelay_SHC(IN := FALSE);
			ELSE
				stat.sState := CONCAT('LN2 low level at SHA. SHC start timeout: ',
							 F_TON_TO_TIME_STRING(Timer := tDelay_SHC));
			END_IF
			IF ctrl.bReset THEN
				stat.nStandAloneFillingState := E_MET_CRYO_LN2_FILLING_STATE.CHECK_PRECONDITIONS;
			END_IF
			
		(**** Begin LN2 control at SHC (Bottom Segment) ****)			
			
		E_MET_CRYO_LN2_FILLING_STATE.START_LEVEL_CONTROL_SHC:

			IF lc_ln2_level_ctrl[3].out_LN2_Level = E_METIS_CRYO_LN2_SENSOR_LEVELS.LOW OR 
				lc_ln2_level_ctrl[3].out_LN2_Level = E_METIS_CRYO_LN2_SENSOR_LEVELS.HIGH OR
				lc_ln2_level_ctrl[3].out_LN2_Level = E_METIS_CRYO_LN2_SENSOR_LEVELS.HIGH_ALARM THEN
				
				stat.nStandAloneFillingState := E_MET_CRYO_LN2_FILLING_STATE.LEVEL_LOW_SHC;
				stat.sState := 'LN2 at or above low level at SHC';
			ELSE
				
				stat.sState := 'Filling Stiff Ring + Bottom segment...';
							
			END_IF
			IF ctrl.bReset THEN
				stat.nStandAloneFillingState := E_MET_CRYO_LN2_FILLING_STATE.CHECK_PRECONDITIONS;
			END_IF
			
		(**** LN2 reached low level at SHC ****)

		E_MET_CRYO_LN2_FILLING_STATE.LEVEL_LOW_SHC:

			tDelay_SHB(IN := TRUE, PT := tDelaySHB);
			IF tDelay_SHB.Q THEN

				stat.nStandAloneFillingState := E_MET_CRYO_LN2_FILLING_STATE.START_LEVEL_CONTROL_SHB;
				tDelay_SHB(IN := FALSE);
			ELSE
				stat.sState := CONCAT('LN2 low level at SHC. SHB start timeout: ',
							 F_TON_TO_TIME_STRING(Timer := tDelay_SHB));
			END_IF
			IF ctrl.bReset THEN
				stat.nStandAloneFillingState := E_MET_CRYO_LN2_FILLING_STATE.CHECK_PRECONDITIONS;
			END_IF

		(**** Begin LN2 control at SHB (Middle Segment) ****)	
			
		E_MET_CRYO_LN2_FILLING_STATE.START_LEVEL_CONTROL_SHB:
		
			// Start Middle Segment Fill (SHB)
			ctrl.bEnable_LN2_Level_Control[2] := TRUE;
			stat.sState := 'Filling Middle Segment...';
			stat.nStandAloneFillingState := E_MET_CRYO_LN2_FILLING_STATE.FILLING;
			
			IF ctrl.bReset THEN
				stat.nStandAloneFillingState := E_MET_CRYO_LN2_FILLING_STATE.CHECK_PRECONDITIONS;
			END_IF

		(**** Actively filling LN2 (steady operation) ****)
		
		E_MET_CRYO_LN2_FILLING_STATE.FILLING:
		
			IF NOT in_Cryo_Stat.bEvacuationActive THEN
				M_SetError(E1004_PumpsNotRunning, 'Evacuation is not active');
				stat.nStandAloneFillingState := E_MET_CRYO_LN2_FILLING_STATE.ERROR;
			ELSIF NOT bESO_LN2_Supply THEN
				M_SetError(E1005_LN2SupplyNotReady, 'LN2 Supply is not available');
				stat.nStandAloneFillingState := E_MET_CRYO_LN2_FILLING_STATE.ERROR;
			ELSE
				
				IF in_Cryo_Stat.lrRadiationShieldsTempK > in_lrRadShld_TempK_TO_Start_PTCs THEN
					stat.sState := CONCAT('Filling All Vessels – Waiting Shields Temp <', LREAL_TO_STRING(in_lrRadShld_TempK_TO_Start_PTCs));
//					IF NOT M_Check_LN2_Filling_Status() THEN
//						RETURN; // Error detected or recovery in progress
//					END_IF

				ELSE
						stat.nStandAloneFillingState := E_MET_CRYO_LN2_FILLING_STATE.RADIATION_SHIELDS_COLD;
				END_IF

			IF ctrl.bReset THEN
				stat.nStandAloneFillingState := E_MET_CRYO_LN2_FILLING_STATE.CHECK_PRECONDITIONS;
			END_IF					
			
			END_IF

		(**** Shield are COLD enough ****)			
			
		E_MET_CRYO_LN2_FILLING_STATE.RADIATION_SHIELDS_COLD:
		
			IF NOT lc_ln2_level_ctrl[1].bActive THEN
					ctrl.bEnable_LN2_Level_Control[1] := TRUE;
			END_IF
			
			IF NOT lc_ln2_level_ctrl[2].bActive THEN
					ctrl.bEnable_LN2_Level_Control[2] := TRUE;
			END_IF
			
			IF NOT lc_ln2_level_ctrl[1].bActive THEN
					ctrl.bEnable_LN2_Level_Control[2] := TRUE;
			END_IF		
			
			M_Standalone_LN2_Filling := TRUE; // Allow sequence to continue
			IF ctrl.bReset THEN
				stat.nStandAloneFillingState := E_MET_CRYO_LN2_FILLING_STATE.NONE;
			END_IF
					
	
		E_MET_CRYO_LN2_FILLING_STATE.ERROR: // Error Handling / Safe Shutdown
			IF ctrl.bReset THEN
				stat.nStandAloneFillingState := E_MET_CRYO_LN2_FILLING_STATE.NONE;
			END_IF
			IF NOT M_Check_LN2_Filling_Status() THEN
				RETURN; // Error detected or recovery in progress
			END_IF
			// Optional: auto-reset if conditions restored
			IF in_Cryo_Stat.bEvacuationActive AND bESO_LN2_Supply THEN
				stat.nStandAloneFillingState := E_MET_CRYO_LN2_FILLING_STATE.NONE;
			END_IF
	
		END_CASE

ELSE
	stat.nStandAloneFillingState := E_MET_CRYO_LN2_FILLING_STATE.CHECK_PRECONDITIONS;
	ctrl.bEnable_LN2_Level_Control[1] := FALSE;
	ctrl.bEnable_LN2_Level_Control[2] := FALSE;
	ctrl.bEnable_LN2_Level_Control[3] := FALSE;
	
	tDelay_SHB(IN := FALSE);
	tDelay_SHC(IN := FALSE);
	
	M_Activity_Stop_LN2_Filling();

END_IF
END_METHOD

(*Cool_Down*)
METHOD M_StateMachine
VAR_INPUT
END_VAR
VAR_IN_OUT
	{attribute 'OPC.UA.DA' := '0'}
	all_cryo_temps:					FB_METIS_TEMPERATURES;
	{attribute 'OPC.UA.DA' := '0'}
	all_heaters:					FB_METIS_HEATERS;
	{attribute 'OPC.UA.DA' := '0'}
	all_t_ctrls:      				FB_METIS_TCTRL;
	{attribute 'OPC.UA.DA' := '0'}
	all_t_votes: 					FB_METIS_VOTERS;
	{attribute 'OPC.UA.DA' := '0'}
	interlocks:						T_METIS_CRYO_INTERLOCKS;
END_VAR


//--- State Machine Logic ---
CASE stat.nState OF
	

	E_MET_CRYO_COOLDOWN_STATE.NONE:
	
		M_Activity_None(
						all_cryo_temps:= all_cryo_temps,
						all_heaters := all_heaters,
						all_t_ctrls := all_t_ctrls,
						all_t_votes := all_t_votes,
						interlocks := interlocks);
						
	E_MET_CRYO_COOLDOWN_STATE.CHECK_PRECONDITIONS:
	
		M_Activity_Check_Preconditions();
	
	E_MET_CRYO_COOLDOWN_STATE.START_COOL_DOWN:
	
		M_Activity_Start_Cool_Down(
									all_cryo_temps:= all_cryo_temps,
									all_heaters := all_heaters,
									all_t_ctrls := all_t_ctrls,
									all_t_votes := all_t_votes,
									interlocks := interlocks);
									
	E_MET_CRYO_COOLDOWN_STATE.START_FILLING_LN2:
	
		M_Activity_Start_LN2_Filling(
									all_cryo_temps:= all_cryo_temps,
									all_heaters := all_heaters,
									all_t_ctrls := all_t_ctrls,
									all_t_votes := all_t_votes,
									interlocks := interlocks);
		
	E_MET_CRYO_COOLDOWN_STATE.START_PTCS:
		M_Activity_Start_PTCs(
									all_cryo_temps:= all_cryo_temps,
									all_heaters := all_heaters,
									all_t_ctrls := all_t_ctrls,
									all_t_votes := all_t_votes,
									interlocks := interlocks);
	E_MET_CRYO_COOLDOWN_STATE.START_TEMP_CTRL_PTC:
	
		M_Activity_Start_Temp_Ctrl_PTC(
									all_cryo_temps:= all_cryo_temps,
									all_heaters := all_heaters,
									all_t_ctrls := all_t_ctrls,
									all_t_votes := all_t_votes,
									interlocks := interlocks);
	E_MET_CRYO_COOLDOWN_STATE.KEEP_COOLING:
	
			M_Activity_Keep_Cooling(
									all_cryo_temps:= all_cryo_temps,
									all_heaters := all_heaters,
									all_t_ctrls := all_t_ctrls,
									all_t_votes := all_t_votes,
									interlocks := interlocks);
		
	E_MET_CRYO_COOLDOWN_STATE.STOPPING_COOL_DOWN:
	
		M_Activity_Stopping_Cool_Down(
									all_cryo_temps:= all_cryo_temps,
									all_heaters := all_heaters,
									all_t_ctrls := all_t_ctrls,
									all_t_votes := all_t_votes,
									interlocks := interlocks);
		
	E_MET_CRYO_COOLDOWN_STATE.FINISHED:
	
		M_Activity_Cool_Down_Finished();
		
	E_MET_CRYO_COOLDOWN_STATE.ERROR:
	
		M_Activity_Error_Handling();


END_CASE;
END_METHOD

METHOD M_Stop_PTCs_During_WarmUP : BOOL
VAR_INPUT
END_VAR
VAR_INST
	
END_VAR
IF in_Cryo_Stat.bStop_PTCs AND in_Cryo_Stat.bWarmUpActive THEN
	M_Activity_Stop_PTCs();
END_IF
END_METHOD

METHOD M_UpdateStatus
VAR_INPUT
END_VAR
VAR_IN_OUT
	{attribute 'OPC.UA.DA' := '0'}
	all_cryo_temps:					FB_METIS_TEMPERATURES;
	{attribute 'OPC.UA.DA' := '0'}
	all_heaters:					FB_METIS_HEATERS;
	{attribute 'OPC.UA.DA' := '0'}
	all_t_ctrls:      				FB_METIS_TCTRL;
	{attribute 'OPC.UA.DA' := '0'}
	all_t_votes: 					FB_METIS_VOTERS;
	{attribute 'OPC.UA.DA' := '0'}
	interlocks:						T_METIS_CRYO_INTERLOCKS;
END_VAR


// References are set once the evacuation system is configured.
IF stat.bConfigured	THEN
	//stat.bRootPumpON	:= rpRef.M_IsReady();
	//stat.bTurboPumpON	:= tpRef.M_IsReady();
END_IF


out_bCoolDownActive := stat.bActive;
stat.bBusy := stat.bActive;

// Check Pre-Conditions for HMI Enable 


stat.bPreConditionsMet := 	in_Cryo_Stat.bInVacuum 	 				AND
							NOT in_Cryo_Stat.bWarmUpActive  		AND
							in_Cryo_Stat.bVentingValvesAreClosed    AND
							NOT in_Cryo_Stat.bRegenerationActive 	AND
							in_Cryo_Stat.bPumpsAreRunning 	 		AND
							bESO_LN2_Supply;
							
M_Check_Is_ReadyForOperation(		all_cryo_temps:= all_cryo_temps,
									all_heaters := all_heaters,
									all_t_ctrls := all_t_ctrls,
									all_t_votes := all_t_votes,
									interlocks := interlocks);
// LN2 level control Timers' times									
									
tEarlyRefillTotal := REAL_TO_TIME(lrEarlyRefillTotal * 3600000.0);  // Hours
tEarlyRefillCycle := REAL_TO_TIME(lrEarlyRefillCycle * 3600000.0);  // Hours

tDelaySHB:= REAL_TO_TIME(lrDelaySHB * 1000.0);  // Seconds
tDelaySHC := REAL_TO_TIME(lrDelaySHC * 1000.0);  // Seconds
tDelaySHCold:= REAL_TO_TIME(lrDelaySHCold *  3600000.0); // Hours
END_METHOD

END_FUNCTION_BLOCK

// POUs/Devices/LN2_Level_Ctrl/FB_METIS_CRYO_LN2_LEVEL_CTRL
	{attribute 'TcHmiSymbol.Show'}
FUNCTION_BLOCK  FB_METIS_CRYO_LN2_LEVEL_CTRL
VAR_INPUT
	in_sName:				STRING;
	in_bEnable:				BOOL;
	{attribute 'TcHmiSymbol.Show'}
	in_ESO_LN2_Supply:		BOOL := TRUE; // Status of LN2 supply from ESO
	in_LN2_TimeOut:			TIME := T#120M;
	in_bEarly_Refilling:	BOOL := FALSE;
	
END_VAR
VAR_OUTPUT
	out_LN2_Level:		E_METIS_CRYO_LN2_SENSOR_LEVELS:= E_METIS_CRYO_LN2_SENSOR_LEVELS.NO_LN2;			
END_VAR
VAR
	{attribute 'TcHmiSymbol.Show'}
	LN2_Level:			FB_METIS_CRYO_LN2_SENSOR;
	{attribute 'TcHmiSymbol.Show'}
	LN2_Valve:			FB_CRYO_VALVE_CTRL;
	{attribute 'TcHmiSymbol.Show'}
	cfg: 				T_LN2_LEVEL_CTRL_CFG;
	{attribute 'OPC.UA.DA' := '1'}
	{attribute 'TcHmiSymbol.Show'}
    ctrl:        		T_LN2_LEVEL_CTRL_CTRL;
	
	LN2_Absent_Timer : TON;
	
	lrEarly_LN2_Refilling_TempK: 		LREAL := 96.0;
	lrEarlyRefilling_Stop_TempK:		LREAL:= 85.0;
	// stat
	bConfigured: 		BOOL := FALSE;
	{attribute 'TcHmiSymbol.Show'}	
	sState:				STRING(80);
	{attribute 'TcHmiSymbol.Show'}
	sSubState:			STRING(80);
	{attribute 'TcHmiSymbol.Show'}
	bError:				BOOL := FALSE;
	{attribute 'TcHmiSymbol.Show'}
	bReset:				BOOL := FALSE;
	{attribute 'TcHmiSymbol.Show'}
	nState: 			E_LN2_LEVEL_CTRL_STATE := E_LN2_LEVEL_CTRL_STATE.OFF; // for state machine
	{attribute 'TcHmiSymbol.Show'}
	bActive: 			BOOL := FALSE;
	{attribute 'TcHmiSymbol.Show'}
	bAuto:				BOOL := TRUE;
	{attribute 'TcHmiSymbol.Show'}
	bManual:			BOOL := FALSE;
	{attribute 'TcHmiSymbol.ShowRecursively'}
	{attribute 'TcHmiSymbol.ReadOnly'}
	stAlarms:		T_CRYO_ALARMS;
	
	// ctrl
	{attribute 'TcHmiSymbol.Show'}
	bEnable:			BOOL := FALSE; // Enable the automatic control
	{attribute 'TcHmiSymbol.Show'}
	bEarly_Refilling:	BOOL := TRUE; // Always atart with Enable early refilling
	bEnable_Valve: 		BOOL;   // Enable flag for the valve
		// Command Override
	{attribute 'TcHmiSymbol.Show'}
	cor_ln2_level_ctrl:	FB_CRYO_CMD_OVERRIDE;
	
	// Timers
	
	// When Cooldown starts, LN2 level control not wait for the LOW sensor before starting the refilling
	TimeOut_LN2_Early_Refill_Duration: 	TON;
	tEarly_Refill_Duration_Time: 		TIME := T#24H;
	bEnable_EarlyRefillingTimer:		BOOL := FALSE;
	
	// During Early refill, Refilling will restart after tCycle_Time
	TimeOut_Early_Refill_Cycle:		 	TON;
	tCycle_Time: 						TIME := T#2H;
	bToggleCycleTimer:					BOOL:= FALSE;
	
	{attribute 'OPC.UA.DA' := '0'}
	{attribute 'TcHmiSymbol.Show'}
    fbConfig    : FB_READ_WRITE_LN2_LEVEL_CONTROL_CONFIG; 
	
	// Triggers.
	//
	// Capture Enable/Disable.
	trigEnable:		R_TRIG;	// bEnable_met_evac
	trigDisable:	F_TRIG;	// bEnable_met_evac
	
	// State-machine vars
	bInit_Filling: BOOL := FALSE;
	{attribute 'TcHmiSymbol.Show'}
	bFilling:						BOOL := TRUE; // Flag to stop filling when level is high and Start at low-Alarm
    nValveResetAttempts : USINT := 0;   // 0..5 attempts
	tonLevelInvalid : TON; // 2-minute timer
	timeLevelInvalidRecovery: TIME := T#2M; 
	
				// Alarm handling
	// List of alarms to be handled by Temperature
	arrEventEntry : ARRAY [0..5] OF TcEventEntry;
	// Alarm handler FB
	fbAlarmHandler : FB_AlarmHandler;
	{attribute 'TcHmiSymbol.Show'}
	{attribute 'TcHmiSymbol.ReadOnly'}
	sInstanceName : T_MaxString;
	{attribute 'TcHmiSymbol.Show'}
	bConfirmAllAlarms : BOOL;
	{attribute 'TcHmiSymbol.Show'}
	{attribute 'TcHmiSymbol.ReadOnly'}
	sEventClassName : T_MaxString;
	
	// Logs logs
	logs:	FB_CRYO_FUNCTION_LOG;	
	
	
END_VAR


// Read/write the configuration
fbConfig(in_sLN2LevelCtrlName:= in_sName, cfg := cfg);


IF bAuto THEN
	bEnable := in_bEnable;
	bEarly_Refilling := in_bEarly_Refilling;
ELSIF bManual THEN
	;
END_IF

bEarly_Refilling := FALSE; // Early Refilling at this level is disabled


M_Configure();

M_ReadSensors();

M_HandleEvents();

M_ExecuteControllers();


M_UpdateStatus();

M_StateMachine();

// read/write the config (if needed)
M_Read_Write_Config();



// Handle alarms
M_UpdateAlarms();

METHOD M_Activity_CheckPreConditions : BOOL
VAR_INPUT
END_VAR
	
IF bEnable THEN
	

	M_Activity_CheckPreConditions := FALSE;
	
	// Handle valve error 
	IF LN2_Valve.stat.bError THEN
		// If we have retries left, attempt reset
		IF nValveResetAttempts < 5 THEN
			LN2_Valve.M_Reset(); // One reset attempt
			nValveResetAttempts := nValveResetAttempts + 1;
	
			bError := FALSE;
			sState := CONCAT('Valve Error - resetting (attempt ',
		CONCAT(USINT_TO_STRING(nValveResetAttempts), '/5)') );
			RETURN;       
		ELSE
			// Max retries exceeded -> error state 99
			bError := TRUE;
			sState := 'Valve Error - max reset attempts exceeded';
			nState := E_LN2_LEVEL_CTRL_STATE.ERROR; // Error State
			RETURN;
		END_IF
	ELSE
		// No valve error
		nValveResetAttempts := 0;
	END_IF
	
	// Other error conditions (sensor, supply, etc.)
	IF NOT LN2_Level.stat.bValid THEN
		bError := TRUE;
		sState := 'Faulty Sensor';
		nState := E_LN2_LEVEL_CTRL_STATE.ERROR; // Error State
		RETURN;
	END_IF
	
	IF NOT in_ESO_LN2_Supply THEN
		bError := TRUE;
		sState := 'LN2 Supply OFF';
		nState := E_LN2_LEVEL_CTRL_STATE.ERROR; // Error State
		RETURN;
	END_IF
	
	IF LN2_Valve.stat.bCtrlOK AND LN2_Level.stat.bValid THEN
		bError := FALSE;
	
		IF bEarly_Refilling THEN
			nState := E_LN2_LEVEL_CTRL_STATE.EARLY_REFILLING;  // Move to Early Refilling
			sState := 'Early Refilling';
		ELSE
			nState := E_LN2_LEVEL_CTRL_STATE.LEVEL_MONITORING; // Level monitoring
			sState := 'Level Monitoring';
		END_IF
	
		M_Activity_CheckPreConditions := TRUE; 
	ELSE
		// Fallback: controller not OK or other unexpected combination
		bError := TRUE;
		sState := 'Preconditions not met (Controller or Level invalid)';
		nState := E_LN2_LEVEL_CTRL_STATE.ERROR;
		M_Activity_CheckPreConditions := FALSE;
	END_IF
	
	
	bFilling := TRUE;
	
ELSE
	
	nState := E_LN2_LEVEL_CTRL_STATE.OFF;    // Move to OFF

    // bFilling := FALSE;
	bEnable_Valve := FALSE;
    bToggleCycleTimer := FALSE;
    bEnable_EarlyRefillingTimer := FALSE;

    TimeOut_LN2_Early_Refill_Duration(
        IN := bEnable_EarlyRefillingTimer,
        PT := tEarly_Refill_Duration_Time
    );
    TimeOut_Early_Refill_Cycle(
        IN := bToggleCycleTimer,
        PT := tCycle_Time
    );

    sState := 'LN2 Level Control OFF';
    sSubState := '';
	
END_IF
END_METHOD

METHOD M_Activity_EarlyRefilling : BOOL
VAR_INPUT
END_VAR
IF bEnable THEN
	// Control LN2 Filling (base logic)
	M_FillingControl();
	
	// Early refilling active
	IF bEarly_Refilling THEN
	
		// Start 24hrs timer once level is high
		IF LN2_Level.out_nLN2_level = E_METIS_CRYO_LN2_SENSOR_LEVELS.HIGH THEN
			
			// Enable 24h early-refill timer only once
			IF NOT bEnable_EarlyRefillingTimer THEN
				bEnable_EarlyRefillingTimer := TRUE;
			END_IF
	
			// Enable 2h cycle timer during early refilling
			bToggleCycleTimer := TRUE;
	
			// Stop filling
			bFilling := FALSE;
		END_IF
	
		// 24 hrs Early refilling Timer
		TimeOut_LN2_Early_Refill_Duration(
			IN := bEnable_EarlyRefillingTimer,
			PT := tEarly_Refill_Duration_Time
		);
	
		// Early refilling period still active?
		IF NOT TimeOut_LN2_Early_Refill_Duration.Q THEN
	
			// Status with remaining time
			sState := CONCAT('LN2 early refilling: ',
							 F_TON_TO_TIME_STRING(Timer := TimeOut_LN2_Early_Refill_Duration));
	
			// 2 hrs filling cycle timer during early refilling
			TimeOut_Early_Refill_Cycle(
				IN := bToggleCycleTimer,
				PT := tCycle_Time
			);
	
			IF TimeOut_Early_Refill_Cycle.Q THEN
				// After 2 hours, start a refill cycle
				bToggleCycleTimer := FALSE;       // reset 2h timer for next cycle
				TimeOut_Early_Refill_Cycle(
					IN := bToggleCycleTimer,
					PT := tCycle_Time
				);
				bFilling := TRUE;                 // Start filling
				sSubState := 'Refilling cycle: active';
			ELSE
				// Waiting for next early refilling cycle
				//bFilling := FALSE;                // Stop filling
				sSubState := CONCAT('Refilling cycle: ',
									F_TON_TO_TIME_STRING(Timer := TimeOut_Early_Refill_Cycle));
				
				// during 2 hours if LN2 drops to LOW-ALARM, start filling again					
				IF LN2_Level.out_nLN2_level = E_METIS_CRYO_LN2_SENSOR_LEVELS.LOW_ALARM THEN					
					bToggleCycleTimer := FALSE;       // reset 2h timer for next cycle
					TimeOut_Early_Refill_Cycle(
						IN := bToggleCycleTimer,
						PT := tCycle_Time
					);
					bFilling := TRUE;                 // Start filling
					sSubState := 'Refilling cycle: active';
				END_IF					
										
				
			END_IF
	
		ELSE
			// 24h early-refilling period finished
			nState := E_LN2_LEVEL_CTRL_STATE.LEVEL_MONITORING;                         // Move to level monitoring
	
			// Cleanup timers and flags
		   // bFilling := FALSE;
			bToggleCycleTimer := FALSE;
			bEnable_EarlyRefillingTimer := FALSE;
	
			bEarly_Refilling := FALSE;
			
			TimeOut_LN2_Early_Refill_Duration(
				IN := bEnable_EarlyRefillingTimer,
				PT := tEarly_Refill_Duration_Time
			);
			TimeOut_Early_Refill_Cycle(
				IN := bToggleCycleTimer,
				PT := tCycle_Time
			);
	
			sState := 'LN2 early refilling: completed';
			sSubState := '';
		END_IF
	
	ELSE
		// Early refilling disabled from HMI -> ensure clean exit
	
		nState := E_LN2_LEVEL_CTRL_STATE.LEVEL_MONITORING;                             // Move to level monitoring
	
		// bFilling := FALSE;
		bToggleCycleTimer := FALSE;
		bEnable_EarlyRefillingTimer := FALSE;
	
		TimeOut_LN2_Early_Refill_Duration(
			IN := bEnable_EarlyRefillingTimer,
			PT := tEarly_Refill_Duration_Time
		);
		TimeOut_Early_Refill_Cycle(
			IN := bToggleCycleTimer,
			PT := tCycle_Time
		);
	
		sState := 'LN2 early refilling: disabled';
		sSubState := '';
	END_IF

ELSE
	
	nState := E_LN2_LEVEL_CTRL_STATE.OFF;    // Move to OFF

    // bFilling := FALSE;
	bEnable_Valve := FALSE;
    bToggleCycleTimer := FALSE;
    bEnable_EarlyRefillingTimer := FALSE;

    TimeOut_LN2_Early_Refill_Duration(
        IN := bEnable_EarlyRefillingTimer,
        PT := tEarly_Refill_Duration_Time
    );
    TimeOut_Early_Refill_Cycle(
        IN := bToggleCycleTimer,
        PT := tCycle_Time
    );

    sState := 'LN2 Level Control OFF';
    sSubState := '';
	
END_IF
END_METHOD

METHOD M_Activity_ErrorHandeling : BOOL
VAR_INPUT
END_VAR
IF bEnable THEN


	bEnable_Valve := FALSE;
	bError := TRUE;
	M_ResetValve();
	
	
	//add error handling if needed.
	IF bReset THEN
		bError := FALSE;
		bReset := FALSE;
	//	bEarly_Refilling := TRUE;
		bFilling := TRUE;
		nState := E_LN2_LEVEL_CTRL_STATE.CHECK_PRECONDITIONS;
		LN2_Valve.M_Reset();
		    // bFilling := FALSE;
		bEnable_Valve := FALSE;
    	bToggleCycleTimer := FALSE;
    	bEnable_EarlyRefillingTimer := FALSE;

		TimeOut_LN2_Early_Refill_Duration(
			IN := bEnable_EarlyRefillingTimer,
			PT := tEarly_Refill_Duration_Time
		);
		TimeOut_Early_Refill_Cycle(
			IN := bToggleCycleTimer,
			PT := tCycle_Time
		);
		
		
	ELSE
		nState := E_LN2_LEVEL_CTRL_STATE.ERROR;
	END_IF

ELSE
	
	nState := E_LN2_LEVEL_CTRL_STATE.OFF;    // Move to OFF

    // bFilling := FALSE;
	bEnable_Valve := FALSE;
    bToggleCycleTimer := FALSE;
    bEnable_EarlyRefillingTimer := FALSE;

    TimeOut_LN2_Early_Refill_Duration(
        IN := bEnable_EarlyRefillingTimer,
        PT := tEarly_Refill_Duration_Time
    );
    TimeOut_Early_Refill_Cycle(
        IN := bToggleCycleTimer,
        PT := tCycle_Time
    );

    sState := 'LN2 Level Control OFF';
    sSubState := '';
	
END_IF
END_METHOD

METHOD M_Activity_Level_Monitoring : BOOL
VAR_INPUT
END_VAR
IF bEnable THEN
	
	M_Activity_Level_Monitoring := FALSE;
	
	// 1) Base filling control (handles sensor validity, NO_LN2 timeout, etc.)
	IF NOT M_FillingControl() THEN
		// Assume M_FillingControl sets bError, sState, nState appropriately
		// Do not overwrite sState / sSubState here
		RETURN;
	END_IF
	
	// Early refilling NOT Active  -> pure level monitoring
	IF NOT bEarly_Refilling THEN
	
		// Make sure early-refilling timers are not running anymore
		bToggleCycleTimer := FALSE;
		bEnable_EarlyRefillingTimer := FALSE;
	
		TimeOut_LN2_Early_Refill_Duration(
			IN := FALSE,
			PT := tEarly_Refill_Duration_Time
		);
		TimeOut_Early_Refill_Cycle(
			IN := FALSE,
			PT := tCycle_Time
		);
	
		sState    := 'LN2 level control active';
		sSubState := 'Level monitoring';
	
		M_Activity_Level_Monitoring := TRUE;
	
	ELSE
		// Early refilling Enabled from HMI -> ensure clean exit
	
		nState := E_LN2_LEVEL_CTRL_STATE.EARLY_REFILLING;  
	
		bToggleCycleTimer := FALSE;
		bEnable_EarlyRefillingTimer := FALSE;
	
		// 
		TimeOut_LN2_Early_Refill_Duration(
			IN := FALSE,
			PT := tEarly_Refill_Duration_Time
		);
		TimeOut_Early_Refill_Cycle(
			IN := FALSE,
			PT := tCycle_Time
		);
	
		sState    := 'LN2 early refilling: Enabled';
		sSubState := '';
	
		M_Activity_Level_Monitoring := TRUE;
	END_IF


ELSE
	
	nState := E_LN2_LEVEL_CTRL_STATE.OFF;    // Move to OFF

    // bFilling := FALSE;
	bEnable_Valve := FALSE;
    bToggleCycleTimer := FALSE;
    bEnable_EarlyRefillingTimer := FALSE;

    TimeOut_LN2_Early_Refill_Duration(
        IN := bEnable_EarlyRefillingTimer,
        PT := tEarly_Refill_Duration_Time
    );
    TimeOut_Early_Refill_Cycle(
        IN := bToggleCycleTimer,
        PT := tCycle_Time
    );

    sState := 'LN2 Level Control OFF';
    sSubState := '';
	
END_IF
END_METHOD

METHOD M_Check_LN2_Level : BOOL
//VAR_INPUT
//END_VAR
//VAR_INST
//	bHA:		BOOL;
//	bH:			BOOL;
//	bL:			BOOL;
//	bLA:		BOOL;
//END_VAR
//CASE LN2_Level.out_nLN2_level OF
//	E_METIS_CRYO_LN2_SENSOR_LEVELS.LOW_ALARM:
//		bEnable_Valve := TRUE;
//		sState := 'LN2 Filling Active';
//	E_METIS_CRYO_LN2_SENSOR_LEVELS.LOW:
//		bL := TRUE;
//	E_METIS_CRYO_LN2_SENSOR_LEVELS.HIGH:
//		bH := TRUE;
//	E_METIS_CRYO_LN2_SENSOR_LEVELS.HIGH_ALARM:
//		bEnable_Valve := FALSE;
//		sState := 'LN2 Level High Alarm';
//	E_METIS_CRYO_LN2_SENSOR_LEVELS.NO_LN2:
//		// Wait for liquiq Nitrogen for in_LN2_TimeOut time after LN2 supply is ON  
//		LN2_Absent_Timer(IN:= TRUE, PT := in_LN2_TimeOut);
//			IF LN2_Absent_Timer.Q THEN
//				 bEnable_Valve := FALSE;
//				 bError := TRUE;
//				 sState	:= 'LN2 Detection Time-out';
//				 bActive := FALSE;
//			ELSE 
//				 bEnable_Valve := TRUE;
//				 sState := 'LN2 Filling Active';
//				 nState := 10; // Active State
//				 bActive := TRUE;
//			END_IF
		
//	E_METIS_CRYO_LN2_SENSOR_LEVELS.Error:
//		bError := TRUE;
//		nState := 99; // Error State
//		sState := 'Faulty Sensor';
//		bActive := FALSE;
//	ELSE
//		bEnable_Valve := FALSE;
//END_CASE


//IF (NOT bHA) OR (NOT bH) THEN
//	bEnable_Valve := TRUE;
//	sState := 'Filling LN2...';

//END_IF
END_METHOD

METHOD M_Configure
VAR_INPUT
END_VAR
VAR_INST
    {attribute 'OPC.UA.DA' := '0'}
    nConfigureState : INT;
END_VAR
arrEventEntry[0] := Tc_Events.METISCryoLN2LevelCtrlEventClass.LevelSensorInvalid;
arrEventEntry[1] := Tc_Events.METISCryoLN2LevelCtrlEventClass.LN2DetectionTimeout;
arrEventEntry[2] := Tc_Events.METISCryoLN2LevelCtrlEventClass.ValveError;
arrEventEntry[3] := Tc_Events.METISCryoLN2LevelCtrlEventClass.LN2SupplyNotReady;
arrEventEntry[4] := Tc_Events.METISCryoLN2LevelCtrlEventClass.LevelLowAlarm;
arrEventEntry[5] := Tc_Events.METISCryoLN2LevelCtrlEventClass.LevelHighAlarm;


IF NOT bConfigured	THEN
	
CASE nConfigureState OF
    0:         
        // start reading the config
        fbConfig.M_ReadConfiguration();
        nConfigureState := 1;
    1:
        IF fbConfig.bReadingDoneFlag THEN           
            // clear the flag
            fbConfig.M_ClearReadingDoneFlag();          

        END_IF
END_CASE

	bConfigured	:= TRUE;;
ELSE
	RETURN;	// Nothing to do any more
END_IF
END_METHOD

METHOD M_ExecuteControllers
VAR_INPUT
END_VAR
//
// Specific Cryo Lab Evacuation System HW configuration.
//

// Valve

cor_ln2_level_ctrl(in_bEnable:= bEnable_Valve);

LN2_Valve(
	in_bEnable		:= cor_ln2_level_ctrl.out_bEnable,
	in_nFeedback	:= E_CRYO_BIN_ACT_FEEDBACK.ON_ONLY);
END_METHOD

METHOD M_FillingControl : BOOL
VAR_INPUT
	
END_VAR
//VAR_INST
//	bfilling_Init:	BOOL := FALSE;
//END_VAR

M_FillingControl := FALSE;

// Level validity with 2-minute delay to error
IF NOT LN2_Level.stat.bValid THEN
    tonLevelInvalid(IN := TRUE, PT := timeLevelInvalidRecovery);

    IF tonLevelInvalid.Q THEN
        // After timeout -> Error
        bError := TRUE;
        sState := 'Faulty Sensor (timeout)';
        nState := E_LN2_LEVEL_CTRL_STATE.ERROR;       // Error State
        bActive := FALSE;
        bEnable_Valve := FALSE;
    ELSE
        // Waiting -> no error yet
        bError := FALSE;
        sState := 'Waiting: Level sensor invalid';
        bActive := FALSE;
        bEnable_Valve := FALSE;
    END_IF

    // In both cases, control is not OK yet
    M_FillingControl := FALSE;
    RETURN;
END_IF

// Sensor valid -> reset invalid-sensor timer
tonLevelInvalid(IN := FALSE);

// Level Control

bError := FALSE;  // clear previous errors

CASE LN2_Level.out_nLN2_level OF

    (****** LOW_ALARM ******)
    E_METIS_CRYO_LN2_SENSOR_LEVELS.LOW_ALARM:
        sState := 'LN2 level ≥ Low-Alarm threshold';
        bEnable_Valve := TRUE;
        bActive := TRUE;
        bFilling := TRUE;

    (****** LOW ******)
    E_METIS_CRYO_LN2_SENSOR_LEVELS.LOW:
        sState := 'LN2 level ≥ Low threshold';
        bEnable_Valve := bFilling;
        bActive := TRUE;

    (****** HIGH ******)
    E_METIS_CRYO_LN2_SENSOR_LEVELS.HIGH:
        sState := 'LN2 level ≥ High threshold';
        bActive := TRUE;
        bEnable_Valve := FALSE;
        bFilling := FALSE;

    (****** HIGH_ALARM ******)
    E_METIS_CRYO_LN2_SENSOR_LEVELS.HIGH_ALARM:
		sState := 'LN2 level ≥ High-Alarm threshold';
        bEnable_Valve := FALSE;
        bActive := TRUE;
        bFilling := FALSE;

    (****** NO_LN2 ******)
    E_METIS_CRYO_LN2_SENSOR_LEVELS.NO_LN2:
        // drive timer on NO_LN2, else reset below
        LN2_Absent_Timer(IN := TRUE, PT := in_LN2_TimeOut);

        IF LN2_Absent_Timer.Q THEN
            bEnable_Valve := FALSE;
            bError := TRUE;
            sState := 'LN2 Detection Time-out';
            bActive := FALSE;
            nState := E_LN2_LEVEL_CTRL_STATE.ERROR; // Error State
        ELSE
            bEnable_Valve := TRUE;
            sState := 'LN2 Filling Active';
            bActive := TRUE;
			bFilling := TRUE;
        END_IF

    (****** Error ******)
    E_METIS_CRYO_LN2_SENSOR_LEVELS.Error:
        bError := TRUE;
        nState := E_LN2_LEVEL_CTRL_STATE.ERROR; // Error State
        sState := 'Faulty Sensor';
        bActive := FALSE;
        bEnable_Valve := FALSE;
		bFilling := FALSE;

END_CASE

// Reset NO_LN2 timer when not in that state
IF LN2_Level.out_nLN2_level <> E_METIS_CRYO_LN2_SENSOR_LEVELS.NO_LN2 THEN
    LN2_Absent_Timer(IN := FALSE);
END_IF


M_FillingControl := NOT bError;
END_METHOD

METHOD M_HandleEvents
VAR_INPUT
END_VAR
VAR_INST
    nEvacOnOffState : UINT := 0; // 0=Idle, 10=AutoOn, 20=AutoOff, 30=ManualOn, 40=ManualOff
END_VAR



trigEnable  (CLK := bEnable);
trigDisable (CLK := bEnable);


IF trigEnable.Q THEN
	M_ResetValve();
END_IF

IF trigDisable.Q THEN
	M_ResetValve();
END_IF
END_METHOD

METHOD M_Read_Write_Config
VAR_INPUT
END_VAR
VAR_IN_OUT
END_VAR

IF ctrl.bWriteConfig THEN
    
    // (update the cfg object if needed)
    // ...
    
    // write the cfg object
    fbConfig.M_WriteConfiguration();
    ctrl.bWriteConfig := FALSE;
            
ELSIF ctrl.bReadConfig THEN

    fbConfig.M_ReadConfiguration();
    ctrl.bReadConfig := FALSE;
    
END_IF


IF fbConfig.bReadingDoneFlag THEN
    // clear the flag
    fbConfig.M_ClearReadingDoneFlag();
END_IF
END_METHOD

METHOD M_ReadSensors : BOOL
VAR_INPUT
END_VAR

// LN2_Level(in_sName:= );

 LN2_Level(
	out_nLN2_level=> , 
	out_bValid=> , 
	out_lrTSensTempK_HA=> , 
	out_lrTSensTempK_H=> , 
	out_lrTSensTempK_L=> , 
	out_lrTSensTempK_LA=> , 
	in_sName:= in_sName,  
	in_lr_LN2Level_Hold_Time:= 			cfg.lr_LN2Level_Hold_Time, 
	in_lrLN2_Level_SenseTempK_HA:= 		cfg.lrLN2_Level_SenseTempK_HA, 
	in_lrLN2_Level_SenseTempK_H:= 		cfg.lrLN2_Level_SenseTempK_H, 
	in_lrLN2_Level_SenseTempK_L:= 		cfg.lrLN2_Level_SenseTempK_L, 
	in_lrLN2_Level_SenseTempK_LA:= 		cfg.lrLN2_Level_SenseTempK_LA, 
	in_lrLN2_Level_AbsenceTempK_HA:= 	cfg.lrLN2_Level_AbsenceTempK_HA, 
	in_lrLN2_Level_AbsenceTempK_H:= 	cfg.lrLN2_Level_AbsenceTempK_H, 
	in_lrLN2_Level_AbsenceTempK_L:= 	cfg.lrLN2_Level_AbsenceTempK_L, 
	in_lrLN2_Level_AbsenceTempK_LA:= 	cfg.lrLN2_Level_AbsenceTempK_LA);
END_METHOD

METHOD M_Reset : BOOL
VAR_INPUT
END_VAR
bReset := TRUE;
END_METHOD

METHOD M_ResetValve : BOOL
VAR_INPUT
END_VAR
LN2_Valve.M_Reset();
END_METHOD

METHOD M_Set_LN2FillingFlag : BOOL
VAR_INPUT
END_VAR
bFilling := TRUE;
END_METHOD

METHOD M_StateMachine
VAR_INST

END_VAR

CASE nState OF

	E_LN2_LEVEL_CTRL_STATE.OFF:
	
		IF bEnable THEN
			bActive := TRUE;
			nState := E_LN2_LEVEL_CTRL_STATE.CHECK_PRECONDITIONS;
		ELSE
			sState := 'OFF';
			nState := 0; // 
			bActive := FALSE;
			bError := FALSE;
			sState := 'OFF';
			bEnable_Valve := FALSE;
			// Reset timer
			LN2_Absent_Timer(IN:= FALSE);
		END_IF
	
	E_LN2_LEVEL_CTRL_STATE.CHECK_PRECONDITIONS: // Initial State: Check configuration and sensor validity
		
		M_Activity_CheckPreConditions();
	
	E_LN2_LEVEL_CTRL_STATE.EARLY_REFILLING: // Early refilling for tLN2_Refill_Early_Start_Time time

		M_Activity_EarlyRefilling();
		
	E_LN2_LEVEL_CTRL_STATE.LEVEL_MONITORING: // Level Monitoring
	
		M_Activity_Level_Monitoring();
		
	E_LN2_LEVEL_CTRL_STATE.ERROR:	// Error State
	
		M_Activity_ErrorHandeling();
		
		
END_CASE
END_METHOD

METHOD M_UpdateAlarms
VAR_INPUT
END_VAR
VAR
	stEventEntry : TcEventEntry;
	sText : STRING;
	
	bValveError : BOOL;
END_VAR
// Valve error summary
bValveError := LN2_Valve.stat.bError;


//
// Set / clear alarms
//

// 0 - LN2 level sensor invalid
fbAlarmHandler.M_UpdateAlarm(
    in_bCondition    := NOT LN2_Level.stat.bValid,
    in_nIndex        := 0,
    in_strEventEntry := Tc_Events.METISCryoLN2LevelCtrlEventClass.LevelSensorInvalid
);


// 1 - LN2 detection timeout
fbAlarmHandler.M_UpdateAlarm(
    in_bCondition    := LN2_Absent_Timer.Q,
    in_nIndex        := 1,
    in_strEventEntry := Tc_Events.METISCryoLN2LevelCtrlEventClass.LN2DetectionTimeout
);


// 2 - LN2 valve error
fbAlarmHandler.M_UpdateAlarm(
    in_bCondition    := bValveError,
    in_nIndex        := 2,
    in_strEventEntry := Tc_Events.METISCryoLN2LevelCtrlEventClass.ValveError
);


// 3 - LN2 supply not ready
fbAlarmHandler.M_UpdateAlarm(
    in_bCondition    := NOT in_ESO_LN2_Supply,
    in_nIndex        := 3,
    in_strEventEntry := Tc_Events.METISCryoLN2LevelCtrlEventClass.LN2SupplyNotReady
);


// 4 - LN2 low alarm level
fbAlarmHandler.M_UpdateAlarm(
    in_bCondition    := LN2_Level.out_nLN2_level = E_METIS_CRYO_LN2_SENSOR_LEVELS.LOW_ALARM,
    in_nIndex        := 4,
    in_strEventEntry := Tc_Events.METISCryoLN2LevelCtrlEventClass.LevelLowAlarm
);


// 5 - LN2 high alarm level
fbAlarmHandler.M_UpdateAlarm(
    in_bCondition    := LN2_Level.out_nLN2_level = E_METIS_CRYO_LN2_SENSOR_LEVELS.HIGH_ALARM,
    in_nIndex        := 5,
    in_strEventEntry := Tc_Events.METISCryoLN2LevelCtrlEventClass.LevelHighAlarm
);


//
// Handle alarms
//
fbAlarmHandler(stAlarms := stAlarms);

fbAlarmHandler.M_ProcessAlarms(
    arrEventEntry := arrEventEntry,
    sEventString  := in_sName
);
END_METHOD

METHOD M_UpdateStatus
VAR_INPUT
END_VAR



out_LN2_Level:= LN2_Level.out_nLN2_level;


tEarly_Refill_Duration_Time := LREAL_TO_TIME(cfg.lr_Early_Refill_Duration_Time * 60.0 * 60.0 * 1000.0);

tCycle_Time := LREAL_TO_TIME(cfg.lr_Cycle_Time * 60.0 * 60.0 * 1000.0);


// Alarm Handeling

sInstanceName := fbAlarmHandler.sInstanceName;
sEventClassName := fbAlarmHandler.sEventClassName;
IF bConfirmAllAlarms THEN
	bConfirmAllAlarms := FALSE;
	fbAlarmHandler.M_ConfirmAllAlarms();
END_IF
END_METHOD

END_FUNCTION_BLOCK

// POUs/Devices/LN2_Level_Sensor/FB_METIS_CRYO_LN2_SENSOR
//
// This FB reads the level of LN2 using four temperature sensors, i.e. instances of FB_CRYO_PT100.
// The resulting level value is the number of temperature sensors showing temperature below in_lrLN2_Temp.
// Provides status of each sensor.
//
{attribute 'TcHmiSymbol.Show'}
FUNCTION_BLOCK FB_METIS_CRYO_LN2_SENSOR
VAR_OUTPUT
	out_nLN2_level: E_METIS_CRYO_LN2_SENSOR_LEVELS := E_METIS_CRYO_LN2_SENSOR_LEVELS.Error;
	out_bValid: 	BOOL := TRUE;
	
	out_lrTSensTempK_HA:		LREAL;
	out_lrTSensTempK_H:			LREAL;
	out_lrTSensTempK_L:			LREAL;
	out_lrTSensTempK_LA:		LREAL;
END_VAR
VAR_INPUT
	
	{attribute 'OPC.UA.DA' := '0'}
	in_sName:				STRING	:=	''; 
	{attribute 'OPC.UA.DA' := '0'}
	in_bSimulation:			BOOL	:= FALSE;	// If TRUE, the temperature value is simulated.
	
	in_lr_LN2Level_Hold_Time:	LREAL := 20.0;
	
	// Threshold temperature read by the heated pt100s when submerged under LN2
	in_lrLN2_Level_SenseTempK_HA:		LREAL;
	in_lrLN2_Level_SenseTempK_H:		LREAL;
	in_lrLN2_Level_SenseTempK_L:		LREAL;
	in_lrLN2_Level_SenseTempK_LA:		LREAL;

// Threshold temperature read by the heated pt100s when LN2 is absent OR Evaporated 
	
	in_lrLN2_Level_AbsenceTempK_HA:		LREAL;
	in_lrLN2_Level_AbsenceTempK_H:		LREAL;
	in_lrLN2_Level_AbsenceTempK_L:		LREAL;
	in_lrLN2_Level_AbsenceTempK_LA:		LREAL;
	
	
END_VAR
VAR
	

	{attribute 'OPC.UA.DA' := '1'}
	Temperature_HA:	FB_CRYO_SENSOR_TEMPERATURE;
	{attribute 'OPC.UA.DA' := '1'}
	Temperature_H:	FB_CRYO_SENSOR_TEMPERATURE;
	{attribute 'OPC.UA.DA' := '1'}
	Temperature_L:	FB_CRYO_SENSOR_TEMPERATURE;
	{attribute 'OPC.UA.DA' := '1'}
	Temperature_LA:	FB_CRYO_SENSOR_TEMPERATURE;
	
	// Four heaters are used to keep pt100 sensors warmer when a sensor is out of LN2.
	// Each heater is connected to a digital OUTPUT. 
	q_bSensorHeaters AT %Q* :	BOOL :=  FALSE;

	{attribute 'OPC.UA.DA' := '1'}
	{attribute 'TcHmiSymbol.Show'}
	stat:			T_METIS_CRYO_LN2_LEVEL_STATUS;
	{attribute 'OPC.UA.DA' := '0'}
	//cfg:			T_METIS_CRYO_LN2_LEVEL_CFG;
	level:			E_METIS_CRYO_LN2_SENSOR_LEVELS := E_METIS_CRYO_LN2_SENSOR_LEVELS.Error;
	
	// Activate heater on the temp sensors
	{attribute 'TcHmiSymbol.Show'}
	bActivateSensor:		BOOL := TRUE;
	
	{attribute 'OPC.UA.DA' := '0'}
	nType_HA:			E_CRYO_SENSOR_TYPE_TEMP	:= E_CRYO_SENSOR_TYPE_TEMP.PT100;
	{attribute 'OPC.UA.DA' := '0'}
	nType_H:				E_CRYO_SENSOR_TYPE_TEMP	:= E_CRYO_SENSOR_TYPE_TEMP.PT100;
	{attribute 'OPC.UA.DA' := '0'}
	nType_L:				E_CRYO_SENSOR_TYPE_TEMP	:= E_CRYO_SENSOR_TYPE_TEMP.PT100;
	{attribute 'OPC.UA.DA' := '0'}
	nType_LA:			E_CRYO_SENSOR_TYPE_TEMP	:= E_CRYO_SENSOR_TYPE_TEMP.PT100;
	
	{attribute 'OPC.UA.DA' := '0'}
	lrScale_HA:			LREAL := 0.1;	// Scale factor, T = raw * scale. Default 0.1
	{attribute 'OPC.UA.DA' := '0'}
	lrScale_H:			LREAL := 0.1;	// Scale factor, T = raw * scale. Default 0.1
	{attribute 'OPC.UA.DA' := '0'}
	lrScale_L:			LREAL := 0.1;	// Scale factor, T = raw * scale. Default 0.1
	{attribute 'OPC.UA.DA' := '0'}
	lrScale_LA:			LREAL := 0.1;	// Scale factor, T = raw * scale. Default 0.1
	
	{attribute 'OPC.UA.DA' := '0'}
	bIgnoreUnderrange_HA:	BOOL := TRUE;	// If True, underrange is also valid
	{attribute 'OPC.UA.DA' := '0'}
	bIgnoreUnderrange_H:		BOOL := TRUE;	// If True, underrange is also valid
	{attribute 'OPC.UA.DA' := '0'}
	bIgnoreUnderrange_L:		BOOL := TRUE;	// If True, underrange is also valid
	{attribute 'OPC.UA.DA' := '0'}
	bIgnoreUnderrange_LA:	BOOL := TRUE;	// If True, underrange is also valid
	{attribute 'OPC.UA.DA' := '0'}
	
	nRampPeriodSec:			UDINT := 60;	// Ramp measurement period [sec]. Default 60 sec.
	
	
	tLN2Level_Hold_Time:	TIME; 

	
END_VAR

// Activate Heaters
M_SetHeatersOutput();

// Get the raw reading and the status of the input channel
M_ReadSensors();

// Calculate temperatures and validity
M_SetStatus();

// Set level and validitiy Outputs
M_SetOutput();

// Get input channel status and the raw reading
METHOD M_ReadSensors
VAR_INPUT
END_VAR
Temperature_HA(	in_nType				:= nType_HA,
				in_lrScale 				:= lrScale_HA, 
				in_bIgnoreUnderrange	:= bIgnoreUnderrange_HA,
				in_nRampPeriodSec		:= nRampPeriodSec);

Temperature_H(	in_nType				:= nType_H,
				in_lrScale 				:= lrScale_H, 
				in_bIgnoreUnderrange	:= bIgnoreUnderrange_H,
				in_nRampPeriodSec		:= nRampPeriodSec);
				                           
Temperature_L(	in_nType				:= nType_L,
				in_lrScale 				:= lrScale_L, 
				in_bIgnoreUnderrange	:= bIgnoreUnderrange_L,
				in_nRampPeriodSec		:= nRampPeriodSec);
                                           
Temperature_LA(	in_nType				:= nType_LA,
				in_lrScale 				:= lrScale_LA, 
				in_bIgnoreUnderrange	:= bIgnoreUnderrange_LA,
				in_nRampPeriodSec		:= nRampPeriodSec);
END_METHOD

METHOD M_SetHeatersOutput
VAR_INPUT
END_VAR
// Turn ON all heaters

IF bActivateSensor THEN
	
q_bSensorHeaters := TRUE;

stat.bActive := TRUE;

ELSE
	
q_bSensorHeaters := FALSE;

stat.bActive := FALSE;

END_IF
END_METHOD

METHOD M_SetOutput : BOOL
VAR_INPUT
END_VAR

out_nLN2_level:= 	level;
out_bValid:=		stat.bValid;


out_lrTSensTempK_HA :=  Temperature_HA.stat.lrTempK;
out_lrTSensTempK_H  :=  Temperature_H.stat.lrTempK;
out_lrTSensTempK_L  :=  Temperature_L.stat.lrTempK;
out_lrTSensTempK_LA :=  Temperature_LA.stat.lrTempK;
END_METHOD

METHOD M_SetStatus
VAR_INPUT
END_VAR
VAR_INST
	bHA, bH, bL, bLA : BOOL;   // Per-level LN2 presence
	
	fbSensor_HA : FB_LN2_LEVEL_PT100_SENSOR;
    fbSensor_H  : FB_LN2_LEVEL_PT100_SENSOR;
    fbSensor_L  : FB_LN2_LEVEL_PT100_SENSOR;
    fbSensor_LA : FB_LN2_LEVEL_PT100_SENSOR;
END_VAR
VAR
    vHA, vH, vL, vLA : BOOL;   // Valid flags
    wHA, wH, wL, wLA : BOOL;   // Warning flags
END_VAR
stat.sName := in_sName;
tLN2Level_Hold_Time := LREAL_TO_TIME(in_lr_LN2Level_Hold_Time * 60.0 * 1000.0);

// --- Evaluate each sensor ---
fbSensor_HA(
    sensor      := Temperature_HA,
    lrSenseTemp := in_lrLN2_Level_SenseTempK_HA,
    lrAbsTemp   := in_lrLN2_Level_AbsenceTempK_HA,
	bPrevPresent:= bHA,
	tHoldTime   := tLN2Level_Hold_Time);
	
	bHA := fbSensor_HA.bLN2Present;
	vHA := fbSensor_HA.bValid;
    wHA := fbSensor_HA.bWarning;
	
fbSensor_H(
    sensor      := Temperature_H,
    lrSenseTemp := in_lrLN2_Level_SenseTempK_H,
    lrAbsTemp   := in_lrLN2_Level_AbsenceTempK_H,
	bPrevPresent:= bH,
	tHoldTime   := tLN2Level_Hold_Time);
	
	bH := fbSensor_H.bLN2Present;
	vH := fbSensor_H.bValid;
	wH := fbSensor_H.bWarning;

fbSensor_L(
    sensor      := Temperature_L,
    lrSenseTemp := in_lrLN2_Level_SenseTempK_L,
    lrAbsTemp   := in_lrLN2_Level_AbsenceTempK_L,
	bPrevPresent:= bL,
	tHoldTime   := tLN2Level_Hold_Time);
	
	bL := fbSensor_L.bLN2Present; 
	vL := fbSensor_L.bValid;
	wL := fbSensor_L.bWarning;

fbSensor_LA(
    sensor      := Temperature_LA,
    lrSenseTemp := in_lrLN2_Level_SenseTempK_LA,
    lrAbsTemp   := in_lrLN2_Level_AbsenceTempK_LA,
	bPrevPresent:= bLA,
	tHoldTime   := tLN2Level_Hold_Time);
	
	bLA := fbSensor_LA.bLN2Present;
	vLA := fbSensor_LA.bValid;
	wLA := fbSensor_LA.bWarning;
	

// Validate all sensors 
IF NOT (vHA AND vH AND vL AND vLA) THEN
    stat.bValid  := FALSE;
    stat.bError  := TRUE;
    stat.sStatus := 'Error: One or more LN2 level sensors invalid';
    RETURN;
END_IF

//  Combine logical states 
IF bLA AND NOT bL AND NOT bH AND NOT bHA THEN
    level := E_METIS_CRYO_LN2_SENSOR_LEVELS.LOW_ALARM;
    stat.sStatus := 'Above Low level alarm';
	
	stat.bLowAlarm 	:= TRUE;
	stat.bLow 		:= FALSE;
	stat.bHigh 		:= FALSE;
	stat.bHighAlarm := FALSE;
	
	stat.bValid  := TRUE;
	stat.bError  := FALSE;

ELSIF bLA AND bL AND NOT bH AND NOT bHA THEN
    level := E_METIS_CRYO_LN2_SENSOR_LEVELS.LOW;
    stat.sStatus := 'Above Low level';
		
	stat.bLowAlarm 	:= TRUE;
	stat.bLow 		:= TRUE;
	stat.bHigh 		:= FALSE;
	stat.bHighAlarm := FALSE;
	
	stat.bValid  := TRUE;
	stat.bError  := FALSE;
	
ELSIF bLA AND bL AND bH AND NOT bHA THEN
    level := E_METIS_CRYO_LN2_SENSOR_LEVELS.HIGH;
    stat.sStatus := 'Above High level';
			
	stat.bLowAlarm 	:= TRUE;
	stat.bLow 		:= TRUE;
	stat.bHigh 		:= TRUE;
	stat.bHighAlarm := FALSE;
	
	stat.bValid  := TRUE;
	stat.bError  := FALSE;

ELSIF bLA AND bL AND bH AND bHA THEN
    level := E_METIS_CRYO_LN2_SENSOR_LEVELS.HIGH_ALARM;
    stat.sStatus := 'Above High level alarm';
	
			
	stat.bLowAlarm 	:= TRUE;
	stat.bLow 		:= TRUE;
	stat.bHigh 		:= TRUE;
	stat.bHighAlarm := TRUE;
	
	stat.bValid  := TRUE;
	stat.bError  := FALSE;

ELSIF NOT bLA AND NOT bL AND NOT bH AND NOT bHA THEN
    level := E_METIS_CRYO_LN2_SENSOR_LEVELS.NO_LN2;
    stat.bError  := TRUE;
    stat.sStatus := 'Error: LN2 not present';
	
			
	stat.bLowAlarm 	:= FALSE;
	stat.bLow 		:= FALSE;
	stat.bHigh 		:= FALSE;
	stat.bHighAlarm := FALSE;
	
	stat.bValid  := TRUE;
	stat.bError  := TRUE;
ELSE
    stat.bValid  := FALSE;
	stat.bError  := TRUE;
    stat.sStatus := 'Faulty sensor combination';
END_IF

// Update warnings per sensor
stat.bWarningSens_HA := wHA;
stat.bWarningSens_H  := wH;
stat.bWarningSens_L  := wL;
stat.bWarningSens_LA := wLA;
END_METHOD

END_FUNCTION_BLOCK

// POUs/Devices/LN2_Level_Sensor/FB_LN2_LEVEL_PT100_SENSOR
FUNCTION_BLOCK FB_LN2_LEVEL_PT100_SENSOR
VAR_INPUT
    sensor        : FB_CRYO_SENSOR_TEMPERATURE;   // PT100 sensor instance
    lrSenseTemp   : LREAL;                         // LN2 present below this temp
    lrAbsTemp     : LREAL;                         // LN2 absent above this temp
    bPrevPresent  : BOOL;                          // Initial last-known state (used on first scan)
    tHoldTime     : TIME;                          // Minimum time to hold "present" after detection
END_VAR
VAR_OUTPUT
    bLN2Present   : BOOL;                          // LN2 detected at this sensor
    bValid        : BOOL;                          // Sensor reading valid
    bWarning      : BOOL;                          // Input over/under warning
END_VAR
VAR
    HoldTimer     : TON;                           // Stability/hold timer
    bInit         : BOOL := TRUE;                  // First-scan initializer
    bHoldActive   : BOOL := FALSE;                 // We are currently enforcing a hold
    bHoldEn       : BOOL := FALSE;                 // TON enable
    bLastPresent  : BOOL := FALSE;                 // Memorized output from previous cycle
END_VAR

//VAR_INPUT
//    sensor       : FB_CRYO_SENSOR_TEMPERATURE;   // PT100 sensor instance
//    lrSenseTemp  : LREAL;                        // LN2 present below this temp
//    lrAbsTemp    : LREAL;                        // LN2 absent above this temp
//	bPrevPresent : BOOL;                		// Last known LN2 state
//	tHoldTime    : TIME;               // How long presence must persist
//END_VAR
//VAR_OUTPUT
//    bLN2Present     : BOOL;                         // LN2 detected at this sensor
//    bValid       : BOOL;                         // Sensor reading valid
//    bWarning     : BOOL;                         // Input over/under warning
//END_VAR
//VAR
//    HoldTimer    : TON;                          // Timer for stability/hysteresis
//END_VAR

//-------------------------------------------------------------------
// One-time initialization: seed the last state from bPrevPresent
//-------------------------------------------------------------------
IF bInit THEN
    bLastPresent := bPrevPresent;
    bLN2Present  := bPrevPresent;
    bInit := FALSE;
END_IF

//-------------------------------------------------------------------
// Default outputs/flags
//-------------------------------------------------------------------
bValid   := FALSE;
bWarning := FALSE;

//-------------------------------------------------------------------
// Validate sensor input first
//-------------------------------------------------------------------
IF sensor.stat.bInputValid AND NOT sensor.stat.bInputOver AND NOT sensor.stat.bInputUnder THEN
    bValid   := TRUE;
    bWarning := FALSE;

    // --- Presence logic with hold ---
    // Start from last known state
    bLN2Present := bLastPresent;

    // Case 1: Temperature indicates LN2 PRESENT immediately
    IF sensor.stat.lrTempK < lrSenseTemp THEN
        // Assert presence now and (re)start hold
        bLN2Present := TRUE;
        bHoldActive := TRUE;

    // Case 2: Temperature indicates LN2 ABSENT (candidate to clear)
    ELSIF sensor.stat.lrTempK > lrAbsTemp THEN
        // Respect hold: only clear after hold time has elapsed
        IF bHoldActive AND (NOT HoldTimer.Q) THEN
            // Still within hold window: keep present
            bLN2Present := TRUE;
        ELSE
            // Hold not active or expired → allow clear
            bLN2Present := FALSE;
            bHoldActive := FALSE;
        END_IF

    // Case 3: Hysteresis band → keep last state. If hold active and not elapsed, keep present.
    ELSE
        IF bHoldActive AND (NOT HoldTimer.Q) THEN
            bLN2Present := TRUE;
        ELSE
            // Keep last state (no change)
            bLN2Present := bLastPresent;
            // release hold after it has elapsed
            IF HoldTimer.Q THEN
                bHoldActive := FALSE;
            END_IF
        END_IF
    END_IF

    // TON enable: run timer whenever we are actively holding and the hold hasn't elapsed yet
    bHoldEn := bHoldActive AND (NOT HoldTimer.Q);

ELSE
    // Sensor invalid → fail-safe
    bValid      := FALSE;
    bWarning    := TRUE;
    bLN2Present := FALSE;
    bHoldActive := FALSE;
    bHoldEn     := FALSE;
END_IF

//-------------------------------------------------------------------
// Run timer EVERY cycle with explicit enable
//-------------------------------------------------------------------
HoldTimer(IN := bHoldEn, PT := tHoldTime);

// Reset timer cleanly when we are not holding
IF NOT bHoldEn THEN
    // Ensures ET resets to T#0 and Q := FALSE as per TON behavior
    HoldTimer(IN := FALSE, PT := tHoldTime);
END_IF

//-------------------------------------------------------------------
// Latch output for next scan
//-------------------------------------------------------------------
bLastPresent := bLN2Present;



//// Default outputs
//bLN2Present := bPrevPresent;

//// Sensor validity check
//IF sensor.stat.bInputValid AND NOT sensor.stat.bInputOver AND NOT sensor.stat.bInputUnder THEN
//    bValid   := TRUE;
//    bWarning := FALSE;

//    // Case 1: LN2 clearly present
//    IF sensor.stat.lrTempK < lrSenseTemp THEN
//        // Immediate reaction
//        bLN2Present := TRUE;

//        // Start hold timer
//        HoldTimer(IN := TRUE, PT := tHoldTime);

//    // Case 2: LN2 clearly absent (and hold expired)
////    ELSIF (sensor.stat.lrTempK > lrAbsTemp) AND (NOT HoldTimer.Q) THEN
//	  ELSIF (sensor.stat.lrTempK > lrAbsTemp) AND ( HoldTimer.Q) THEN
//        HoldTimer(IN := FALSE);
//        bLN2Present := FALSE;

//    // Case 3: Hysteresis / hold zone
//    ELSE
//        // Keep hold active until timer expires
//        IF HoldTimer.Q THEN
//            HoldTimer(IN := FALSE); // Reset after tHoldTime elapsed
//        END_IF;
//        // During hold, bLN2Present stays at previous TRUE state
//        // After timer expired, re-eval will apply on next cycle
//    END_IF

//ELSE
//    // Sensor invalid
//    bValid      := FALSE;
//    bWarning    := TRUE;
//    HoldTimer(IN := FALSE);
//    bLN2Present := FALSE;
//END_IF

//// Save state
//bPrevPresent := bLN2Present;

END_FUNCTION_BLOCK

// POUs/XML_Cfg_Read_Write/FB_READ_WRITE_LN2_LEVEL_CONTROL_CONFIG
FUNCTION_BLOCK FB_READ_WRITE_LN2_LEVEL_CONTROL_CONFIG EXTENDS FB_READ_WRITE_CONFIG_BASE
VAR_INPUT
	in_sLN2LevelCtrlName:      T_MaxString;
END_VAR
VAR_IN_OUT
	cfg:   T_LN2_LEVEL_CTRL_CFG;
END_VAR


	
SUPER^(
    in_sEntryName  := in_sLN2LevelCtrlName,
    in_sSubFolder  := 'LN2Level_Ctrl\',
    in_sXPath      := '/LN2LevelCtrl_Configuration/',
    in_pSymAddr    := ADR(cfg),
    in_cbSymSize   := SIZEOF(cfg));

END_FUNCTION_BLOCK

// POUs/Devices/PTC Cooler/FB_METIS_CRYO_CPA
FUNCTION_BLOCK FB_METIS_CRYO_CPA EXTENDS FB_CRYO_CPA
VAR_INPUT
	{attribute 'OPC.UA.DA' := '0'}
	in_bEnable:						BOOL;			// Flag to Start/Stop PTC
END_VAR
VAR_OUTPUT
END_VAR
VAR
	i_bCompressorRunning  			AT %I*:		BOOL;
	i_bHighPressure  				AT %I*:		BOOL;
	i_bHighTemperature  			AT %I*:		BOOL;
	i_bOK							AT %I*:		BOOL;
END_VAR




IF in_bEnable THEN
	ctrl.nDevCommand := E_CRYO_CPA_CMDS.START;
	ctrl.bExecute := TRUE;

ELSE
	ctrl.nDevCommand := E_CRYO_CPA_CMDS.STOP;
	ctrl.bExecute := TRUE;

END_IF





M_CompressorRunning();
M_HighPressureFlag();
M_HighTemperatureFlag();

// Execute the base FB_CRYO_CPA
SUPER^();

METHOD M_CompressorRunning : BOOL
VAR_INPUT
END_VAR
M_CompressorRunning := i_bCompressorRunning;
END_METHOD

METHOD M_HighPressureFlag : BOOL
VAR_INPUT
END_VAR
M_HighPressureFlag := i_bHighPressure;
END_METHOD

METHOD M_HighTemperatureFlag : BOOL
VAR_INPUT
END_VAR
M_HighTemperatureFlag := i_bHighTemperature;
END_METHOD

END_FUNCTION_BLOCK

// POUs/Functions/F_TIME_HHMMSS
FUNCTION F_TIME_HHMMSS : STRING(16)
VAR_INPUT
END_VAR
VAR
	fbGetSystemTime  : GETSYSTEMTIME;
    fileTime         : T_FILETIME;
    tsTime           : TIMESTRUCT;     // <-- correct type
    sHour, sMin, sSec : STRING(3);
    sTime            : STRING(16);     // result: 'hh:mm:ss'
END_VAR

// Get system time (UTC)
fbGetSystemTime(
    timeLoDW => fileTime.dwLowDateTime,
    timeHiDW => fileTime.dwHighDateTime
);

// Convert FILETIME -> TIMESTRUCT
tsTime := FILETIME_TO_SYSTEMTIME(fileTime);

// ----- Build hh with leading zero -----
IF tsTime.wHour < 10 THEN
    sHour := CONCAT('0', UDINT_TO_STRING(tsTime.whour));
ELSE
    sHour := UDINT_TO_STRING(tsTime.whour);
END_IF

// ----- Build mm with leading zero -----
IF tsTime.wminute < 10 THEN
    sMin := CONCAT('0', UDINT_TO_STRING(tsTime.wminute));
ELSE
    sMin := UDINT_TO_STRING(tsTime.wminute);
END_IF

// ----- Build ss with leading zero -----
IF tsTime.wsecond < 10 THEN
    sSec := CONCAT('0', UDINT_TO_STRING(tsTime.wsecond));
ELSE
    sSec := UDINT_TO_STRING(tsTime.wsecond);
END_IF

// ----- Final string: hh:mm:ss -----
sTime := CONCAT(STR1 := sHour, STR2 := ':');
sTime := CONCAT(STR1 := sTime, STR2 := sMin);
sTime := CONCAT(STR1 := sTime, STR2 := ':');
sTime := CONCAT(STR1 := sTime, STR2 := sSec);

F_TIME_HHMMSS := sTime;

END_FUNCTION

// POUs/Routines/WarmUP/FB_METIS_CRYO_WARM_UP
FUNCTION_BLOCK FB_METIS_CRYO_WARM_UP
VAR_INPUT
	in_sName:							STRING := 'WARM-UP';
	in_Cryo_Stat:						T_METIS_CRYO_STAT;
	in_lrWarmUp_Detectors_Ramp_1:			LREAL := 1.0; // Start detectors warm up with a ramp of 1 K/min
	in_lrWarmUp_Detectors_Ramp_Switch_Temp:	LREAL := 80.0; // ramp switch at 80 K from 1K/min to 6K/h
	in_lrWarmUp_Detectors_Ramp_2:			LREAL := 0.1; // ramp up detectors, new ramp 6 K/h (0.1 K/min)
	in_lrWarmUp_EvacPermission_Temp:		LREAL := 280; // When all temperatures > 280 K,  allow to stop 
	in_lrWarmUp_VentingPermission_Temp:		LREAL := 280; // When all temperatures > 280 K, allow tO start 
	in_lrWarmUp_Alarm_Temp:					LREAL := 310; 
	in_lrWarmUp_Alarm_PreCooling_Pressure:	LREAL := 700; // Pressure precooling system >700 mbar
	// TODO: Detector ramp too fast
	
END_VAR
VAR_OUTPUT
	out_bWarmUpActive:			BOOL := FALSE;
	out_bStop_PTCs:				BOOL := FALSE;
END_VAR
VAR_IN_OUT
	{attribute 'OPC.UA.DA' := '0'}
	all_cryo_temps:					FB_METIS_TEMPERATURES;
	{attribute 'OPC.UA.DA' := '0'}
	all_heaters:					FB_METIS_HEATERS;
	{attribute 'OPC.UA.DA' := '0'}
	all_t_ctrls:      				FB_METIS_TCTRL;
	{attribute 'OPC.UA.DA' := '0'}
	all_t_votes: 					FB_METIS_VOTERS;
	{attribute 'OPC.UA.DA' := '0'}
	interlocks:						T_METIS_CRYO_INTERLOCKS;
END_VAR
VAR	
	sName:				STRING := 'WarmUp_Routine';

	stat:				T_MET_CRYO_WARMUP_STAT;
	ctrl:				T_MET_CRYO_WARMUP_CTRL;
	
	
	// Triggers
		//
	// Capture Enable/Disable.
	trigEnable:		R_TRIG;	// in_bEnable
	trigDisable:	F_TRIG;	// in_bEnable
	
	
	// Events Handleing
	
	arrEventEntry : ARRAY [0..6] OF TcEventEntry;
	// Alarm handler FB
	fbAlarmHandler : FB_AlarmHandler;
	
	stAlarms:		T_CRYO_ALARMS;

	/////////////////////
	// Cryo System logs
	/////////////////////
		
	logs:	FB_CRYO_FUNCTION_LOG;
END_VAR
VAR CONSTANT

    // --- [3000] Preconditions ---
    E3000_EvacuationNotActive                     : UDINT := 3000001; // Evacuation is not active
    E3001_VentingValveOpen                        : UDINT := 3000002; // Venting valve is not closed
    E3002_LN2RefillingStillActive                 : UDINT := 3000003; // LN2 refilling has not been stopped
    E3003_LN2RefillingNotStopped24hBeforeWarmUp   : UDINT := 3000004; // LN2 refilling was not stopped 24 hours before warm up
    E3004_WarmUpAlreadyActive                     : UDINT := 3000005; // Warm up requested while already active

    // --- [3100] Cooler and Heater Operation Errors ---
    E3100_CoolersFailedToStop                     : UDINT := 3100001; // One or more coolers failed to stop
    E3101_DetectorWarmUpHeaterFailed              : UDINT := 3100002; // Detector warm-up heater failed
    E3102_SubsystemWarmUpHeaterFailed             : UDINT := 3100003; // Warm-up heater of a cold subsystem failed
    E3103_RadiationShieldHeaterFailed             : UDINT := 3100004; // Radiation shield heater failed
    E3104_TemperatureControlFailedToStart         : UDINT := 3100005; // Temperature control failed to start
    E3105_TemperatureControlFailedToStop          : UDINT := 3100006; // Temperature control failed to stop
    E3106_WarmUpHeaterShutdownTimeout             : UDINT := 3100007; // One or more heaters remained active during shutdown

    // --- [3200] Temperature Monitoring Errors ---
    E3200_DetectorRampTooFast                     : UDINT := 3200001; // Detector temperature ramp exceeds allowed rate
    E3201_DetectorDidNotReach80K                  : UDINT := 3200002; // Detector did not reach 80 K within expected time
    E3202_RadiationShieldWarmUpNotStarted         : UDINT := 3200003; // Radiation shield warm up did not start when detectors were > 80 K
    E3203_SubsystemRampTooFast                    : UDINT := 3200004; // One or more cold subsystems warmed faster than allowed
    E3204_TemperatureTooHigh                      : UDINT := 3200005; // One or more temperatures > 310 K
    E3205_TemperatureSensorFault                  : UDINT := 3200006; // One or more temperature sensors invalid or faulty
    E3206_TemperatureNotRising                    : UDINT := 3200007; // Temperature did not increase as expected during warm up
    E3207_NotAllTemperaturesAbove280K             : UDINT := 3200008; // Not all required temperatures are above 280 K
    E3208_DetectorWarmUpRampControlFault          : UDINT := 3200009; // Detector ramp control failed or unstable
    E3209_SubsystemWarmUpControlFault             : UDINT := 3200010; // Subsystem warm-up control failed or unstable

    // --- [3300] Pressure Monitoring Errors ---
    E3300_PrecoolingPressureTooHigh               : UDINT := 3300001; // Pressure in precooling system > 700 mbar
    E3301_CryostatPressureRiseUnexpected          : UDINT := 3300002; // Unexpected pressure increase during warm up
    E3302_EvacuationPressureNotSafeForStop        : UDINT := 3300003; // Pressure not safe to allow evacuation stop

    // --- [3400] Sequence Timing Errors ---
    E3400_StopCoolersTimeout                      : UDINT := 3400001; // Coolers did not stop within allowed time
    E3401_DetectorRampTo80KTimeout                : UDINT := 3400002; // Detector ramp to 80 K exceeded allowed time
    E3402_WarmUpTo280KTimeout                     : UDINT := 3400003; // Warm up to 280 K exceeded allowed time
    E3403_WarmUpTo290KTimeout                     : UDINT := 3400004; // Warm up to 290 K exceeded allowed time
    E3404_WarmUpSequenceTimeout                   : UDINT := 3400005; // Entire warm-up sequence exceeded maximum duration

    // --- [3500] Manual Intervention / Abort ---
    E3500_OperatorAbortedWarmUp                   : UDINT := 3500001; // Operator manually stopped warm up
    E3501_OperatorStoppedHeatersDuringWarmUp      : UDINT := 3500002; // Operator stopped one or more heaters during warm up
    E3502_OperatorChangedControlMode              : UDINT := 3500003; // Operator changed temperature control unexpectedly

    // --- [3600] Interlock Violations ---
    E3600_VentingRequestedBelow280K               : UDINT := 3600001; // Venting requested while one or more temperatures < 280 K
    E3601_PrecoolingActiveDuringWarmUp            : UDINT := 3600002; // Precooling system active during warm up
    E3602_CoolerStartRequestedDuringWarmUp        : UDINT := 3600003; // Cooler start requested while warm up is active
    E3603_EvacuationStopRequestedBelow280K        : UDINT := 3600004; // Evacuation stop requested before all temperatures > 280 K

    // --- [3700] Shutdown / Recovery Failures ---
    E3700_WarmUpHeatersDidNotDisable              : UDINT := 3700001; // Warm-up heaters failed to disable during stop
    E3701_TemperatureControlStillActiveAfterStop  : UDINT := 3700002; // Temperature control remained active after stop command
    E3702_WarmUpShutdownTimeout                   : UDINT := 3700003; // Warm-up shutdown did not complete in time

END_VAR




M_Configure();


M_StateMachine(all_cryo_temps:= all_cryo_temps,
						all_heaters := all_heaters,
						all_t_ctrls := all_t_ctrls,
						all_t_votes := all_t_votes,
						interlocks := interlocks);

M_UpdateStatus();

M_HandleEvents();

METHOD M_Activity_Check_Preconditions
VAR_INPUT
END_VAR

// CHECK_WARMUP_PRECONDITIONS

stat.bActive := TRUE;
stat.bBusy := FALSE; 
stat.bDone := FALSE;  

// --- Precondition Check: Venting Valves Closed ---
IF NOT in_Cryo_Stat.bVentingValvesAreClosed THEN
    stat.nState := E_MET_CRYO_WARMUP_STATE.ERROR;
    stat.sState := 'Error: Venting valves are not closed.';
    RETURN; 
END_IF

// --- Precondition Check: Pumps Running ---
IF NOT in_Cryo_Stat.bEvacuationActive THEN
    stat.nState := E_MET_CRYO_WARMUP_STATE.ERROR;
    stat.sState := 'Error: Pumps are not running.';
    RETURN; 
END_IF

// --- Precondition Check: Cool Down Active ---
IF in_Cryo_Stat.bCoolDownActive THEN
    stat.nState := E_MET_CRYO_WARMUP_STATE.ERROR;
    stat.sState := 'Error: Cool down is active.';
    RETURN; 
END_IF

stat.nState := E_MET_CRYO_WARMUP_STATE.START_WARM_UP;
stat.sState := 'Preconditions met. Starting warm-up.';
END_METHOD

METHOD M_Activity_Error_Handling
VAR_INPUT
END_VAR
VAR_IN_OUT
	{attribute 'OPC.UA.DA' := '0'}
	all_cryo_temps:					FB_METIS_TEMPERATURES;
	{attribute 'OPC.UA.DA' := '0'}
	all_heaters:					FB_METIS_HEATERS;
	{attribute 'OPC.UA.DA' := '0'}
	all_t_ctrls:      				FB_METIS_TCTRL;
	{attribute 'OPC.UA.DA' := '0'}
	all_t_votes: 					FB_METIS_VOTERS;
	{attribute 'OPC.UA.DA' := '0'}
	interlocks:						T_METIS_CRYO_INTERLOCKS;
END_VAR
stat.bActive := TRUE;
in_cryo_stat.bPermitEvacuationStop := FALSE; // Evacuation cannot stop, yet


IF NOT ctrl.bEnable THEN
	all_heaters.h_cry_sha.M_SetDisable();
	all_heaters.h_cry_shb.M_SetDisable();
	all_heaters.h_cry_shc.M_SetDisable();

	all_t_ctrls.tc_cry_sha.M_SetDisable();
	all_t_ctrls.tc_cry_shb.M_SetDisable();
	all_t_ctrls.tc_cry_shc.M_SetDisable();
	
	stat.sState := 'Deactivating all heaters';
	stat.nState := E_MET_CRYO_WARMUP_STATE.NONE;
END_IF




IF ctrl.bReset THEN 
	stat.nState := E_MET_CRYO_WARMUP_STATE.NONE;
	ctrl.bReset := FALSE;
	ctrl.bEnable := FALSE;						// Disable Regeneration
END_IF
END_METHOD

METHOD M_Activity_Finished
VAR_INPUT
END_VAR


stat.bActive := FALSE;
stat.bBusy := FALSE;
stat.bDone := TRUE;

stat.nState := E_MET_CRYO_WARMUP_STATE.NONE;

logs.M_LogInfo('Warm_Up finished');
END_METHOD

METHOD M_Activity_Keep_Ramping_Up_Detectors
VAR_INPUT
END_VAR
stat.nState := E_MET_CRYO_WARMUP_STATE.RAMP_UP_DETECTORS_6K;
END_METHOD

METHOD M_Activity_Keep_Warming_Up
VAR_INPUT
END_VAR
VAR_IN_OUT
	{attribute 'OPC.UA.DA' := '0'}
	all_cryo_temps:					FB_METIS_TEMPERATURES;
END_VAR
// TODO implement the activity


IF NOT trigDisable.Q THEN 
	


	IF in_Cryo_Stat.lrHighestTempK < in_lrWarmUp_EvacPermission_Temp THEN
		stat.nState := 	E_MET_CRYO_WARMUP_STATE.KEEP_WARMING_UP;
		stat.sState := 'Warming Up ...';
		logs.M_LogInfo('Warming Up ...');
	ELSE
		stat.nState := E_MET_CRYO_WARMUP_STATE.STOPPING_WARM_UP;
		logs.M_LogInfo('Warm_UP temperature achieved...');
		logs.M_LogInfo('Warm_UP stopped automatically...');
	END_IF
	
	
ELSE

	stat.nState := E_MET_CRYO_WARMUP_STATE.STOPPING_WARM_UP;
	stat.sState := 'Warm_UP interrupted by operator...';
	logs.M_LogInfo('Warm_UP interrupted by operator...');
END_IF
END_METHOD

METHOD M_Activity_None
VAR_INPUT
END_VAR
VAR_IN_OUT
	{attribute 'OPC.UA.DA' := '0'}
	interlocks:						T_METIS_CRYO_INTERLOCKS;
END_VAR
stat.bActive := FALSE;
stat.bError := FALSE;

// Check enable AND Interlocks
IF ctrl.bEnable AND NOT interlocks.bInterlock_WarmUp THEN
	stat.nState := E_MET_CRYO_WARMUP_STATE.CHECK_PRECONDITIONS;
	logs.M_LogInfo('Warm_UP started by operator...');
ELSE
	stat.nState := E_MET_CRYO_WARMUP_STATE.NONE;
	stat.sState := 'Warm_Up OFF';
END_IF
END_METHOD

METHOD M_Activity_Ramp_Up_Detectors_2
VAR_INPUT
END_VAR
// TODO implement the activity

stat.nState := E_MET_CRYO_WARMUP_STATE.START_RAMP_Up_RADIATION_SHIELDS;
END_METHOD

METHOD M_Activity_Start_Ramp_Up_CFO
VAR_INPUT
END_VAR
// TODO implement the activity

stat.nState := E_MET_CRYO_WARMUP_STATE.KEEP_WARMING_UP;
END_METHOD

METHOD M_Activity_Start_Ramp_Up_Detectors_1k
VAR_INPUT
END_VAR
// TODO implement the activity

stat.nState := E_MET_CRYO_WARMUP_STATE.KEEP_RAMPING_Up_DETECTORS;
END_METHOD

METHOD M_Activity_Start_Ramp_Up_IMG
VAR_INPUT
END_VAR
// TODO implement the activity

stat.nState := E_MET_CRYO_WARMUP_STATE.START_RAMP_Up_SCAO;
END_METHOD

METHOD M_Activity_Start_Ramp_Up_LMS
VAR_INPUT
END_VAR
// TODO implement the activity

stat.nState := E_MET_CRYO_WARMUP_STATE.START_RAMP_Up_CFO;
END_METHOD

METHOD M_Activity_Start_Ramp_Up_Radiation_Shields
VAR_INPUT
END_VAR
VAR_IN_OUT
	{attribute 'OPC.UA.DA' := '0'}
	all_cryo_temps:					FB_METIS_TEMPERATURES;
	{attribute 'OPC.UA.DA' := '0'}
	all_heaters:					FB_METIS_HEATERS;
	{attribute 'OPC.UA.DA' := '0'}
	all_t_ctrls:      				FB_METIS_TCTRL;
	{attribute 'OPC.UA.DA' := '0'}
	all_t_votes: 					FB_METIS_VOTERS;
	{attribute 'OPC.UA.DA' := '0'}
	interlocks:						T_METIS_CRYO_INTERLOCKS;
END_VAR


IF NOT trigDisable.Q THEN 
	
		all_heaters.h_cry_sha.M_SetEnable();
		all_heaters.h_cry_shb.M_SetEnable();
		all_heaters.h_cry_shc.M_SetEnable();
		
		all_t_ctrls.tc_cry_sha.M_SetEnable();
		all_t_ctrls.tc_cry_shb.M_SetEnable();
		all_t_ctrls.tc_cry_shc.M_SetEnable();
		
		all_t_ctrls.tc_cry_sha.M_Set_SetPoint(
					m_eSetpointType := E_METIS_CTRL_SETPOINT_SWITCH.FIXED,
					m_lrFixedSetpoint := in_lrWarmUp_EvacPermission_Temp + 10,
					m_lrSetpointOffset := 0.0, 
					m_pSetpointTemp := all_cryo_temps.M_SetTemperatureSensor(0));
					
		all_t_ctrls.tc_cry_shb.M_Set_SetPoint(
					m_eSetpointType := E_METIS_CTRL_SETPOINT_SWITCH.FIXED,
					m_lrFixedSetpoint := in_lrWarmUp_EvacPermission_Temp +10,
					m_lrSetpointOffset := 0.0, 
					m_pSetpointTemp := all_cryo_temps.M_SetTemperatureSensor(0));
					
		all_t_ctrls.tc_cry_shc.M_Set_SetPoint(
					m_eSetpointType := E_METIS_CTRL_SETPOINT_SWITCH.FIXED,
					m_lrFixedSetpoint := in_lrWarmUp_EvacPermission_Temp +10,
					m_lrSetpointOffset := 0.0, 
					m_pSetpointTemp := all_cryo_temps.M_SetTemperatureSensor(0));
		
		stat.nState := E_MET_CRYO_WARMUP_STATE.START_RAMP_Up_IMG;
		stat.sState := 'Heaters and controllers initialized.';
		logs.M_LogInfo('Heaters and temp controls at radiation shields initialized....');	
		
(* 
TODO: Put the Ear-Flange temp control at proper place
////////////Ear Flange temp control //////////////////
*)		
	all_heaters.h_cry_pta.M_SetEnable();
	all_heaters.h_cry_ptb.M_SetEnable();
	all_heaters.h_cry_ptc.M_SetEnable();

	
	all_t_ctrls.tc_cry_pt.M_SetEnable();

	all_t_ctrls.tc_cry_pt.M_Set_SetPoint(
		m_eSetpointType := E_METIS_CTRL_SETPOINT_SWITCH.FIXED,
		m_lrFixedSetpoint := in_lrWarmUp_EvacPermission_Temp + 10.0,
		m_lrSetpointOffset := 0.0, 
		m_pSetpointTemp := all_cryo_temps.M_SetTemperatureSensor(0));
		
				logs.M_LogInfo('Heaters and temp controls at Ear-Flange initialized....');
	
	
ELSE

	stat.nState := E_MET_CRYO_WARMUP_STATE.STOPPING_WARM_UP;
	stat.sState := 'Warm_UP interrupted by operator...';
	logs.M_LogInfo('Warm_UP interrupted by operator...');
END_IF
END_METHOD

METHOD M_Activity_Start_Ramp_Up_SCAO
VAR_INPUT
END_VAR
// TODO implement the activity

stat.nState := E_MET_CRYO_WARMUP_STATE.START_RAMP_Up_LMS;
END_METHOD

METHOD M_Activity_Start_Warm_Up
VAR_INPUT
END_VAR



stat.bPermitEvacuationStop := FALSE; // Evacuation is not allowed to stop
stat.bActive := TRUE;
stat.bBusy := 	TRUE;
stat.bDone := 	FALSE;

stat.nState := E_MET_CRYO_WARMUP_STATE.STOP_PTCs;
END_METHOD

